# B&R Automation Studio project Panasonic_LinkaKapacitorov_A2021040 (part 2)

- Safety project (password-protected, skipped)

### Config.mprecipexml - AB1_CPU/mappServices/Config.mprecipexml
```
Element gRemPremenne (Type=mprecipexml)
```

### Config_1.mprecipexml - AB1_CPU/mappServices/Config_1.mprecipexml
```
Element gUzivatelXmlLink (Type=mprecipexml)
```

### Config_2.mprecipexml - AB1_CPU/mappServices/Config_2.mprecipexml
```
Element gRecipeXmlLink (Type=mprecipexml)
```

## Logical view

Binary libraries used (declarations not repeated): RUNTIME, OPERATOR, AsIecCon, astime, standard, AsBrStr, FileIO, sys_lib, AsSafety, DataObj, AsXml, CoTrace 5.14.0, AsZip, LoopConR 4.10.2, brsystem, dvframe, asstring, AsMath, AsTCP, MpRecipe 5.15.0, MpBase 5.15.0

### Global.typ - Global data types
```iecst
(********************************************************************
 * COPYRIGHT -- Microsoft
 ********************************************************************
 * File: Global.typ
 * Author: Martin
 * Created: February 11, 2016
 ********************************************************************
 * Global data types of project Zamazat_1
 ********************************************************************)
(**************Ovládanie tlačiarne**********************)

TYPE
	Client_typ : 	STRUCT  (*TCP Client Variables*)
		sStep : UINT; (*TCP Client Step Variable*)
		TcpOpen_0 : TcpOpen; (*AsTCP.TcpOpen FUB*)
		TcpClient_0 : TcpClient; (*AsTCP.TcpClient FUB*)
		TcpRecv_0 : TcpRecv; (*AsTCP.TcpRecv FUB*)
		TcpSend_0 : TcpSend; (*AsTCP.TcpSend FUB*)
		TcpIoctl_0 : TcpIoctl; (*AsTCP.TcpIoctl FUB*)
		TcpClose_0 : TcpClose; (*AsTCP.TcpClose FUB*)
		linger_opt : tcpLINGER_typ; (*AsTCP.tcpLINGER_typ*)
		recv_timeout : UDINT; (*receive timeout*)
		TcpOpen_timeout : UDINT;
		TcpClient_timeout : UDINT;
	END_STRUCT;
	Tlaciaren_typ : 	STRUCT
		Commands : TlaciarenCommands_typ;
		Status : TlaciarenStatus_typ;
		Data : TlaciarenData_typ;
	END_STRUCT;
	TlaciarenCommands_typ : 	STRUCT
		PosliSpravu : BOOL;
	END_STRUCT;
	TlaciarenStatus_typ : 	STRUCT
		PoruchaOtvoreniaKomunikacie : BOOL;
		PoruchaOdoslaniaDat : BOOL;
		PoruchaZatvoreniaKomunikacie : BOOL;
		PoruchaSpojenia_s_Tlaciarnou : BOOL;
		PoruchaPrijatiaDat : BOOL;
		PrislaSprava_s_Tlaciarne : BOOL;
	END_STRUCT;
	TlaciarenData_typ : 	STRUCT  (*Datatyp for global Variables*)
		Sprava_pre_Tlaciaren : STRING[4000]; (*Obsahuje posielane data pre tlačiareň v textovej podobe*)
		Odpoved_s_Tlaciarne : STRING[400]; (*Obsahuje odpoveď s tlačiarne*)
	END_STRUCT;
	EtiketaPanasonic_typ : 	STRUCT
		IdentificationNumber : STRING[10];
		ModelType : STRING[8];
		SupplierNumber : STRING[9];
		Country : STRING[2];
		Date : STRING[8];
		Counter : STRING[5];
		DataMetrix : STRING[31];
	END_STRUCT;
END_TYPE

(**********************RFID Čitačky*********************************************)

TYPE
	RFID_typ : 	STRUCT
		IN : RFID_IN_typ;
		OUT : RFID_OUT_typ;
		CMD : RFID_CMD_typ;
		STAV : RFID_STAV_typ;
		PAR : RFID_PAR_typ;
	END_STRUCT;
	RFID_IN_typ : 	STRUCT
		BYTE_IN : ARRAY[0..31]OF USINT;
		Bit_CP : BOOL;
		Bit_AA : BOOL;
		Bit_AE : BOOL;
		Bit_AF : BOOL;
		Bit_MT : BOOL;
		Bit_TO : BOOL;
		Old_Bit_TO : BOOL;
		Bit_HF : BOOL;
		Bit_BB : BOOL;
	END_STRUCT;
	RFID_OUT_typ : 	STRUCT
		BYTE_OUT : ARRAY[0..31]OF USINT;
		Bit_AV : BOOL;
		Bit_GR : BOOL;
		Bit_KA : BOOL;
		Bit_TI : BOOL;
	END_STRUCT;
	RFID_CMD_typ : 	STRUCT
		CitajDATA : BOOL;
		ZapisDATA : BOOL;
		CitaciuHlavu_VYPNI : BOOL;
	END_STRUCT;
	RFID_STAV_typ : 	STRUCT
		CitanieDat_OK : BOOL;
		CitanieDat_ERROR : BOOL;
		ZapisDat_OK : BOOL;
		ZapisDat_ERROR : BOOL;
		PritomnostCipu : BOOL;
	END_STRUCT;
	RFID_PAR_typ : 	STRUCT
		PrecitaneCisloPaletky : STRING[10];
		PrecitanyTypPaletky : STRING[10];
		Zadane_Cislo_Typ_Paletky : STRING[10]; (*Oddelovací znak "bodkočiarka"*)
		Precitane_Cislo_Typ_Paletky : STRING[10];
		PrecitaneCisloPaletky_POLE : ARRAY[0..9]OF USINT;
		ZadaneCisloPaletky_POLE : ARRAY[0..9]OF USINT;
	END_STRUCT;
END_TYPE

(**************************Ručná čitačka QR kódu******************************)

TYPE
	RS232_typ : 	STRUCT
		Command : RS232_Command_typ;
		Status : RS232_Status_typ;
		Step : USINT;
		FRM_xopen_0 : FRM_xopen;
		xopenConfig : XOPENCONFIG;
		FRM_read_0 : FRM_read;
		FRM_write_0 : FRM_write;
		FRM_rbuf_0 : FRM_rbuf;
		FRM_gbuf_0 : FRM_gbuf;
		FRM_robuf_0 : FRM_robuf;
		FRM_close_0 : FRM_close;
		PrecitaneData : STRING[80];
	END_STRUCT;
	RS232_Command_typ : 	STRUCT
		PosielajData : BOOL;
		PrimajData : BOOL;
		ZatvorKomunikaciu : BOOL;
		PotvrdeniePoruchy : BOOL;
	END_STRUCT;
	RS232_Status_typ : 	STRUCT
		PoruchaOtvoreniaKomunikacie : BOOL;
		PoruchaPriradeniaSEND_Buffera : BOOL;
		PoruchaUvolneniaSEND_Buffera : BOOL;
		PoruchaZatvoreniaKomunikacie : BOOL;
		PoruchaCitaniaDat : BOOL;
		PoruchaUvolneniaRECEIVE_Buffera : BOOL;
		PrimanieDat_OK : BOOL;
		PosielanieDat_OK : BOOL;
	END_STRUCT;
END_TYPE

(**************************Remanentne premenné********************************)

TYPE
	RemPremenne_typ : 	STRUCT
		VstupVytah_PozNavazania : UDINT;
		VstupVytah_PozVyvazania : UDINT;
		VystupVytah_PozNavazania : UDINT;
		VystupVytah_PozVyvazania : UDINT;
		PocetDniDoVymenyFiltra : UDINT;
	END_STRUCT;
END_TYPE

(***************Uzivatelia****************************)

TYPE
	ParametreUzivatelovTyp : 	STRUCT
		Meno : STRING[50];
		Heslo : STRING[50];
		UrovenUzivatela : UINT;
	END_STRUCT;
END_TYPE

(************Receptury*************************)

TYPE
	ParametreRecepturTyp : 	STRUCT
		NazovModelu : STRING[18];
		TypPaletky : STRING[4];
		Robot_CisloProgramu : USINT;
		Kamera_CisloProgramuQRkod : USINT;
		Kamera_CisloProgramuDMkod : USINT;
		Robot_PozLepenia_OffsetX : REAL;
		Robot_PozLepenia_OffsetY : REAL;
		Robot_PozLepenia_OffsetZ : REAL;
		RychlostDopravnikaPriCisteni : REAL;
	END_STRUCT;
END_TYPE

(**************************Safety***************************************************)

TYPE
	Safety_typ : 	STRUCT
		IN : Safety_IN_typ;
		OUT : Safety_OUT_typ;
		PAR : Safety_PAR_typ;
		STAV : Safety_STAV_typ;
		RESET_ZonyBunky : BOOL;
		RESET_ZonyCS : BOOL;
		RESET_ZonyVstupnehoVytahu : BOOL;
		RESET_ZonyVystupnehoVytahu : BOOL;
		RESET_DeadMan : BOOL;
		SpatnaVazba_ZonaBunky : BOOL;
		SpatnaVazba_ZonaCS : BOOL;
	END_STRUCT;
	Safety_IN_typ : 	STRUCT
		Robot_CS_CH1 : BOOL;
		Robot_CS_CH2 : BOOL;
		VyblokovanieSafety_CH1 : BOOL;
		VyblokovanieSafety_CH2 : BOOL;
		OvladaciPanel_CS_CH1 : BOOL;
		OvladaciPanel_CS_CH2 : BOOL;
		DopravnikNG_Bariera_CH1 : BOOL;
		DopravnikNG_Bariera_CH2 : BOOL;
		Snimac_ServisneDvere_CH1 : BOOL;
		Snimac_ServisneDvere_CH2 : BOOL;
		ZamkyBunky_CH1 : BOOL;
		ZamkyBunky_CH2 : BOOL;
		MutingRobota_CH1 : BOOL;
		MutingRobota_CH2 : BOOL;
		DeadMan_CH1 : BOOL;
		DeadMan_CH2 : BOOL;
		VstupnyVytah_MutingSnimac_CH1 : BOOL;
		VstupnyVytah_MutingSnimac_CH2 : BOOL;
		VstupnyVytah_Bariera_CH1 : BOOL;
		VstupnyVytah_Bariera_CH2 : BOOL;
		VstupnyVytah_CS_CH1 : BOOL;
		VstupnyVytah_CS_CH2 : BOOL;
		VystupnyVytah_MutingSnimac_CH1 : BOOL;
		VystupnyVytah_MutingSnimac_CH2 : BOOL;
		VystupnyVytah_Bariera_CH1 : BOOL;
		VystupnyVytah_Bariera_CH2 : BOOL;
		VystupnyVytah_CS_CH1 : BOOL;
		VystupnyVytah_CS_CH2 : BOOL;
	END_STRUCT;
	Safety_OUT_typ : 	STRUCT
		Zona_CS : BOOL;
		Zona_Bunky : BOOL;
		Zona_VstupnyVytah : BOOL;
		Zona_VystupnyVytah : BOOL;
	END_STRUCT;
	Safety_PAR_typ : 	STRUCT
		PAR_0 : USINT;
	END_STRUCT;
	Safety_STAV_typ : 	STRUCT
		SafetyPLC_Nabehlo : BOOL;
		ZonaCS_AKTIVNA : BOOL;
		ZonaBunky_Odblokovana : BOOL;
		ZamkyBunky_AKTIVNE : BOOL;
		ZonaBunky_AKTIVNA : BOOL;
		ZonaVstupnyVytah_Odblokovana : BOOL;
		ZonaVstupnyVytah_AKTIVNA : BOOL;
		ZonaVystupnyVytah_Odblokovana : BOOL;
		ZonaVystupnyVytah_AKTIVNA : BOOL;
		BarieraDopravnikaNG_AKTIVNA : BOOL;
		MutingRobota_AKTIVNY : BOOL;
		MutingBarieryVstupVytah_AKTIVNY : BOOL;
		MutingBarieryVystupVytah_AKTIVNY : BOOL;
		BarieraVstupVytahu_AKTIVNA : BOOL;
		BarieraVystupVytahu_AKTIVNA : BOOL;
		ServisneDvereTlaciarne_AKTIVNE : BOOL;
		CS_Robot_Odblokovany : BOOL;
		CS_OvlPanel_Odblokovany : BOOL;
		CS_VstupnyVytah_Odblokovany : BOOL;
		CS_VystupnyVytah_Odblokovany : BOOL;
		VyblokovanieSafety_AKTIVNE : BOOL;
		DeadMan_Odblokovany : BOOL;
		DeadMan_AKTIVNY : BOOL;
	END_STRUCT;
END_TYPE

(**************************Vizualizacia**********************************************)

TYPE
	Vizu_typ : 	STRUCT
		Language_Index : USINT;
		CisloAktualnejObrazovky : USINT;
		CisloZadanejObrazovky : USINT;
		TL_RezimAutomat : BOOL;
		TL_NavratPaletkyNG : BOOL;
		TL_ZamkniPredneDvere : BOOL;
		TL_ZamkniZadneDvere : BOOL;
		StavPracoviskaVstupVytah_Index : USINT;
		StavPracoviskaStopPredCist_Index : USINT;
		StavPracoviskaStopPoCist_Index : USINT;
		StavPracoviskaDoprCistenia_Index : USINT;
		StavPracoviskaStopEtiketov_Index : USINT;
		StavPracoviskaRobota_Index : USINT;
		StavPracoviskaDoprBunky_Index : USINT;
		StavPracoviskaStopDopNG_Index : USINT;
		StavPracoviskaStopVystDopr_Index : USINT;
		StavPracoviskaDoprVystup_Index : USINT;
		StavPracoviskaVystupVytah_Index : USINT;
		StavPracoviskaStopVratDopr_Index : USINT;
		StavPracoviskaDoprVrat_Index : USINT;
		StavZariadenia_Farba : USINT;
		StavZariadenia_Index : USINT;
		StavNGpaletky_Index : USINT;
		StavZmenyModelu_Index : USINT;
		StavZmenyModelu_Farba : USINT;
		TL_ZamokPredneDvere_DISABLE : BOOL;
		TL_ZamokZadneDvere_DISABLE : BOOL;
		TL_RezimManual_DISABLE : BOOL; (*0 - odomknuté, 1 - zamknuté*)
		TL_StartAutomat_DISABLE : BOOL;
		TL_UkoncenieCyklu_DISABLE : BOOL;
		TL_Reset_DISABLE : BOOL;
		TL_ZmenModel_DISABLE : BOOL;
		TL_PotvrdeniePaletky_NG_DISABLE : BOOL;
		TL_ZruseniePaletky_NG_DISABLE : BOOL;
		TL_OdparkujRobota_DISABLE : BOOL;
		ZmenaParametrov_DISABLE : BOOL;
		TL_BunkyRR_DISABLE : BOOL;
		TL_Ovl_Ionizatora_DISABLE : BOOL;
		TL_Ovl_DveriVstupVytahu_DISABLE : BOOL;
		Slider : USINT;
		FarbaTlacitkaAlarm_Index : BOOL;
		FarbaTlacitka_PotvrdPaletkuNG : BOOL;
		FarbaTlacitka_ZamokPredneDvere : USINT;
		FarbaTlacitka_ZamokZadneDvere : USINT;
		ZobrazSymbolAlarmu : BOOL;
		ZobrazHlasenie_ResetZariadenia : USINT;
		ZobrazHlasenie_PotvrdPaletkyNG : USINT;
		ZobrazHlasenie_NespravTypPaletky : USINT;
		ZobrazHlasenie_ZaaretujTlaciaren : USINT;
		ZobrazHlas_ZatvorSerDvereTlac : USINT;
		ZobrazHlasenie_TlaciarenOffline : USINT;
		ZobrazHlasenie_DochadzaPaska : USINT;
		PodsvietenieTlacitka_ResetCS : USINT;
		Nacitany_MODEL : STRING[18];
		Nacitany_LOT : STRING[11];
		NacitanieMODELU_DISABLE : BOOL;
		NacitanieLOTU_DISABLE : BOOL;
		NacitanieMODELU_IndexFarby : USINT;
		NacitanieLOTU_IndexFarby : USINT;
		OverNacitany_MODEL : BOOL;
		OverNacitany_LOT : BOOL;
		TL_VstupVytah_Homing_DISABLE : BOOL;
		TL_VstupVytah_Zdvih_DISABLE : BOOL;
		TL_VstupVytah_Doprav_DISABLE : BOOL;
		TL_VystupVytah_Homing_DISABLE : BOOL;
		TL_VystupVytah_Zdvih_DISABLE : BOOL;
		TL_VystupVytah_Doprav_DISABLE : BOOL;
		TL_Robot_CitanieQRkodu_DISABLE : BOOL;
		TL_Robot_CitanieDMkodu_DISABLE : BOOL;
		TL_Robot_OdoberEtiketu_DISABLE : BOOL;
		ZadavanieKorekciiRobota_DISABLE : BOOL;
		VolbyRezimov_DISABLE : BOOL;
		IndexSuradnicovehoSystemuPaletky : USINT;
		IndexFarbyStavuFiltrov : USINT;
		IndexStavuFiltrov : USINT;
		IndexStavuPasky : USINT;
		IndexStavuLadenieKamery : USINT;
		IndexStavuLadenieKamery_Farba : USINT;
		ZobrazSymbolCS_VstupVytah : USINT;
		ZobrazSymbolCS_VystupVytah : USINT;
		ZobrazSymbolCS_Panel : USINT;
		ZobrazSymbolCS_Robot : USINT;
	END_STRUCT;
END_TYPE

(**************************Linka************************************************)

TYPE
	Linka_typ : 	STRUCT
		IN : Linka_IN_typ;
		OUT : Linka_OUT_typ;
		PAR : Linka_PAR_typ;
		STAV : Linka_STAV_typ;
		Automat : BOOL;
		Manual : BOOL;
		Reset : BOOL;
		KoniecCyklu : BOOL;
		Majak_HukackaON : BOOL;
		CitackaQRkodu_AKTIVNA : BOOL;
		ZmenModel : BOOL;
		VymenaFiltrovPotvrdena : BOOL;
		Rezim_BezTlaceEtikety : BOOL;
		Rezim_BezKomunikacie : BOOL;
		Rezim_BezCistenia : BOOL;
		Rezim_Priechodny : BOOL;
		Rezim_Testovania : BOOL;
		ResetNapajaniaKamery : BOOL;
	END_STRUCT;
	Linka_IN_typ : 	STRUCT
		PrepatovaOchrana_OK : BOOL; (*1 - OK*)
		PoruchaNapajaniaMenicov : BOOL; (*1 - OK*)
		SpatnaVazba_ZonaCS : BOOL; (*1 - OK*)
		SpatnaVazba_ZonaVstupVytah : BOOL; (*1 - OK*)
		SpatnaVazba_ZonaVystupVytah : BOOL; (*1 - OK*)
		SpatnaVazba_ZonaBunky : BOOL; (*1 - OK*)
		SpatnaVazba_VentilTerminal_SQ1 : BOOL;
		SpatnaVazba_VentilTerminal_SQ2 : BOOL;
		PredneDvereZavrete_EZ1 : BOOL;
		ZadneDvereZavrete_EZ2 : BOOL;
		SmartKamera_IN0_CAM1 : BOOL;
		SmartKamera_IN1_CAM1 : BOOL;
		TlakVzduchu_OK_S2 : BOOL;
		IonJednotka_MachineON_RJ1 : BOOL;
		IonJednotka_Error_Sumary_RJ1 : BOOL;
		IonJednotka_Error_Filter1_RJ1 : BOOL;
		IonJednotka_Error_Filter2_RJ1 : BOOL;
		IonJednotka_Error_Motor_RJ1 : BOOL;
		IonJednotka_Error_Network_RJ1 : BOOL;
		IonJednotka_Error_HighVolt_RJ1 : BOOL;
		IonJednotka_Error_ComAirTC1_RJ1 : BOOL;
		IonJednotka_Error_ComAirTC2_RJ1 : BOOL;
		IonJednotka_Error_VolumeFlow_RJ1 : BOOL;
		IonJednotka_Error_TCcontrol_RJ1 : BOOL;
		IonJednotka_Error_Inverter_RJ1 : BOOL;
		IonJednotka_PoruchaNapajania : BOOL;
		SnimacRotacieHornTrysiek_1_IS7 : BOOL;
		SnimacRotacieHornTrysiek_2_IS8 : BOOL;
		SnimacRotacieHornTrysiek_3_IS9 : BOOL;
		SnimacRotacieHornTrysiek_4_IS10 : BOOL;
		SnimacRotacieSpodTrysiek_1_IS11 : BOOL;
		SnimacRotacieSpodTrysiek_2_IS12 : BOOL;
		SnimacRotacieSpodTrysiek_3_IS13 : BOOL;
	END_STRUCT;
	Linka_OUT_typ : 	STRUCT
		Majak_ZeleneSvetlo : BOOL;
		Majak_ZlteSvetlo : BOOL;
		Majak_CerveneSvetlo : BOOL;
		Majak_Hukacka : BOOL;
		PredneDvere_Zamkni_EZ1 : BOOL;
		ZadneDvere_Zamkni_EZ2 : BOOL;
		OsvetlenieBunky_Zapni : BOOL;
		SmartKamera_OUT0_CAM1 : BOOL;
		SmartKamera_OUT1_CAM1 : BOOL;
		VT1_PowerlinkOUTPUTS : ARRAY[0..3]OF USINT;
		IonJednotka_START : BOOL;
		IonJednotka_RESET : BOOL;
		IonJednotka_AIR : BOOL;
		Vzduchotechnika_START : BOOL;
		Rele_ResetNapajaniaKamery : BOOL;
	END_STRUCT;
	Linka_PAR_typ : 	STRUCT
		Zvoleny_MODEL : STRING[18];
		Zvoleny_LOT : STRING[11];
		Zvoleny_TypPaletky : STRING[10];
		IndexZvoleneReceptury : USINT;
		Zvolene_CisloProgramuRobota : USINT;
		Zvolene_KamCisloProg_QRkod : USINT;
		Zvolene_KamCisloProg_DMkod : USINT;
		Zvolena_PozLepenia_OffsetX : REAL;
		Zvolena_PozLepenia_OffsetY : REAL;
		Zvolena_PozLepenia_OffsetZ : REAL;
		Zvolena_RychlostDopravPriCisteni : REAL;
	END_STRUCT;
	Linka_STAV_typ : 	STRUCT
		Automat : BOOL;
		Manual : BOOL;
		PoINIT : BOOL;
		READY_TO_START : BOOL;
		UkoncenieCyklu_BUSY : BOOL;
		Hardware_OK : BOOL;
		PrebiehaZmenaModelu : BOOL;
		PoruchaOtacaniaTrysiek : BOOL;
		FiltreIonizacnejJednotkyZanesene : BOOL;
		IonizacnaJednotka_BUSY : BOOL;
		Dopravniky_PAUZA : BOOL;
	END_STRUCT;
END_TYPE

(**************Stav hardware*****************************)

TYPE
	Hardware_STAV_typ : 	STRUCT
		KartaAB2_ProfinetMaster_OK : BOOL;
		KartaAB3_SafetyMaster_OK : BOOL;
		KartaAB4_SafetyDI_OK : BOOL;
		KartaAB5_16DI_OK : BOOL;
		KartaAB6_16DI_OK : BOOL;
		KartaAB7_16DI_OK : BOOL;
		KartaAB8_16DO_OK : BOOL;
		KartaAB9_16DO_OK : BOOL;
		KartaAB10_X2X_OK : BOOL;
		ModulDI1_16DI_OK : BOOL;
		ModulDI2_16DI_OK : BOOL;
		ModulDI3_8DI_OK : BOOL;
		ModulSI1_4SI_OK : BOOL;
		ModulSI2_4SI_OK : BOOL;
		Komunikacia_Robot_OK : BOOL;
		Komunikacia_Kamera_OK : BOOL;
		Komunikacia_RFIDModul_OK : BOOL;
		Komunikacia_VentTerminal_OK : BOOL;
		Komunikacia_MeniceFM_OK : BOOL;
		Komunikacia_Panasonic_OK : BOOL;
	END_STRUCT;
END_TYPE

(***************VstupnyVytah*************************************)

TYPE
	VstupnyVytah_typ : 	STRUCT
		IN : VstupnyVytah_IN_typ;
		OUT : VstupnyVytah_OUT_typ;
		PAR : VstupnyVytah_PAR_typ;
		STAV : VstupnyVytah_STAV_typ;
		Automat : BOOL;
		Manual : BOOL;
		Reset : BOOL;
		KoniecCyklu : BOOL;
		MenicZdvihu_FM2 : RiadenieFM;
		RR_Dopravnik_VPRED : BOOL;
		RR_Dopravnik_VZAD : BOOL;
	END_STRUCT;
	VstupnyVytah_IN_typ : 	STRUCT
		RiadenieDopravnika_OK_ELR1 : BOOL;
		TeplotaMotora_OK_M1 : BOOL; (*1 - OK*)
		StavMenicaZdvihu_OK_FM2 : BOOL; (*1 - OK*)
		BannerPotvrdeny_IOS1 : BOOL;
		DvereVytahuOtvorene_MS1 : BOOL;
		DvereVytahuZatvorene_MS2 : BOOL;
		PrechodDopravnikaVytahu_OS1 : BOOL;
		PritomnostPaletky_IS3 : BOOL;
		PritomnostProduktu_OS2 : BOOL;
		ReferencnySnimacZdvihu : BOOL; (*Preposielané z FM cez komunikáciu*)
		SpodnyLimitZdvihu : BOOL; (*Preposielané z FM cez komunikáciu*)
		HornyLimitZdvihu : BOOL; (*Preposielané z FM cez komunikáciu*)
	END_STRUCT;
	VstupnyVytah_OUT_typ : 	STRUCT
		Dopravnik_ChodVPRED_ELR1 : BOOL;
		Dopravnik_ChodVZAD_ELR1 : BOOL;
		Banner_ZelenaLED_IOS1 : BOOL;
		Banner_CervenaLED_IOS1 : BOOL;
		DvereVytahu_OTVOR_YV002 : BOOL;
		DvereVytahu_ZATVOR_YV001 : BOOL;
	END_STRUCT;
	VstupnyVytah_PAR_typ : 	STRUCT
		Zdvih_ZadanaPozicia : UDINT;
		Zdvih_ZadanaRychlost : REAL;
		Zdvih_ZadanaJoggRychlost : REAL;
	END_STRUCT;
	VstupnyVytah_STAV_typ : 	STRUCT
		PoINIT : BOOL;
		Zdvih_AktualnaPozicia : UDINT;
		Zdvih_AktualnaRychlost : REAL;
		Zdvih_HomingOK : BOOL;
		Zdvih_BUSY : BOOL;
		Homing_BUSY : BOOL;
		Zdvih_PoziciaDosiahnuta : BOOL;
		PrebiehaVyvazaniePaletky : BOOL;
		VytahNapolohovany : BOOL;
		ObsluhaPotvrdilaBanner : BOOL;
	END_STRUCT;
END_TYPE

(***************StoperPredCistenim*************************************)

TYPE
	StoperPredCistenim_typ : 	STRUCT
		IN : StoperPredCistenim_IN_typ;
		OUT : StoperPredCistenim_OUT_typ;
		PAR : StoperPredCistenim_PAR_typ;
		STAV : StoperPredCistenim_STAV_typ;
		Automat : BOOL;
		Manual : BOOL;
		Reset : BOOL;
		KoniecCyklu : BOOL;
	END_STRUCT;
	StoperPredCistenim_IN_typ : 	STRUCT
		PritomnostPaletky_IS4 : BOOL;
	END_STRUCT;
	StoperPredCistenim_OUT_typ : 	STRUCT
		StoperZASUN_YV005 : BOOL;
	END_STRUCT;
	StoperPredCistenim_PAR_typ : 	STRUCT
		PAR_0 : USINT;
	END_STRUCT;
	StoperPredCistenim_STAV_typ : 	STRUCT
		PoINIT : BOOL;
		PrebiehaVyvazaniePaletky : BOOL;
	END_STRUCT;
END_TYPE

(***************StoperPoCisteni*************************************)

TYPE
	StoperPoCisteni_typ : 	STRUCT
		IN : StoperPoCisteni_IN_typ;
		OUT : StoperPoCisteni_OUT_typ;
		PAR : StoperPoCisteni_PAR_typ;
		STAV : StoperPoCisteni_STAV_typ;
		Automat : BOOL;
		Manual : BOOL;
		Reset : BOOL;
		KoniecCyklu : BOOL;
	END_STRUCT;
	StoperPoCisteni_IN_typ : 	STRUCT
		PritomnostPaletky_IS6 : BOOL;
		ZaplnenieBuffera_IS5 : BOOL;
	END_STRUCT;
	StoperPoCisteni_OUT_typ : 	STRUCT
		StoperZASUN_YV006 : BOOL;
	END_STRUCT;
	StoperPoCisteni_PAR_typ : 	STRUCT
		PAR_0 : USINT;
	END_STRUCT;
	StoperPoCisteni_STAV_typ : 	STRUCT
		PoINIT : BOOL;
		PrebiehaVyvazaniePaletky : BOOL;
	END_STRUCT;
END_TYPE

(***************DopravnikCistenia*************************************)

TYPE
	DopravCistenia_typ : 	STRUCT
		IN : DopravCistenia_IN_typ;
		OUT : DopravCistenia_OUT_typ;
		PAR : DopravCistenia_PAR_typ;
		STAV : DopravCistenia_STAV_typ;
		Automat : BOOL;
		Manual : BOOL;
		Reset : BOOL;
		KoniecCyklu : BOOL;
		MenicDopravnika_FM1 : RiadenieFM;
		RR_Chod_VPRED : BOOL;
		RR_Chod_VZAD : BOOL;
		Dopravnik_RUN : BOOL;
	END_STRUCT;
	DopravCistenia_IN_typ : 	STRUCT
		StavMenica_OK_FM1 : BOOL; (*1 - OK*)
	END_STRUCT;
	DopravCistenia_OUT_typ : 	STRUCT
		New_Member : USINT;
	END_STRUCT;
	DopravCistenia_PAR_typ : 	STRUCT
		ZadanaRychlost : REAL;
		ZadanaJoggRychlost : REAL;
	END_STRUCT;
	DopravCistenia_STAV_typ : 	STRUCT
		PoINIT : BOOL;
		AktualnaRychlost : REAL;
		BUSY : BOOL;
	END_STRUCT;
END_TYPE

(***************DopravnikBunky*************************************)

TYPE
	DopravBunky_typ : 	STRUCT
		IN : DopravBunky_IN_typ;
		OUT : DopravBunky_OUT_typ;
		PAR : DopravBunky_PAR_typ;
		STAV : DopravBunky_STAV_typ;
		Automat : BOOL;
		Manual : BOOL;
		Reset : BOOL;
		KoniecCyklu : BOOL;
	END_STRUCT;
	DopravBunky_IN_typ : 	STRUCT
		RiadenieDopravnika_OK_ELR4 : BOOL;
		TeplotaMotora_OK_M4 : BOOL; (*1 - OK*)
	END_STRUCT;
	DopravBunky_OUT_typ : 	STRUCT
		Dopravnik_ChodVPRED_ELR4 : BOOL;
	END_STRUCT;
	DopravBunky_PAR_typ : 	STRUCT
		PAR_0 : USINT;
	END_STRUCT;
	DopravBunky_STAV_typ : 	STRUCT
		PoINIT : BOOL;
	END_STRUCT;
END_TYPE

(***************StoperEtiketovania*************************************)

TYPE
	StoperEtiketovania_typ : 	STRUCT
		IN : StoperEtiketovania_IN_typ;
		OUT : StoperEtiketovania_OUT_typ;
		PAR : StoperEtiketovania_PAR_typ;
		STAV : StoperEtiketovania_STAV_typ;
		Automat : BOOL;
		Manual : BOOL;
		Reset : BOOL;
		KoniecCyklu : BOOL;
		RR_VytlacEtiketu : BOOL;
		OdosliDataDoPanasonicu : BOOL;
		RR_ZacentrujPaletku : BOOL;
		RR_OdcentrujPaletku : BOOL;
	END_STRUCT;
	StoperEtiketovania_IN_typ : 	STRUCT
		Tlaciaren_KoniecEtikiet : BOOL;
		Tlaciaren_KoniecPasky : BOOL;
		Tlaciaren_Porucha : BOOL;
		Tlaciaren_KoniecTlace : BOOL;
		Tlaciaren_Offline : BOOL;
		Tlaciaren_Dispending : BOOL;
		PritomnostPaletky_IS16 : BOOL;
		Centrovanie_HornaPoloha_IS18 : BOOL;
		Centrovanie_SpodnaPoloha_IS17 : BOOL;
		SuflikTlaciarne_LS_IS23 : BOOL;
		SuflikTlaciarne_PS_IS22 : BOOL;
	END_STRUCT;
	StoperEtiketovania_OUT_typ : 	STRUCT
		Tlaciaren_VytlacEtiketu : BOOL;
		Tlaciaren_VytlacZnovaEtiketu : BOOL;
		Centrovanie_VYSUN_YV003 : BOOL;
		Centrovanie_ZASUN_YV004 : BOOL;
		StoperZASUN_YV007 : BOOL;
	END_STRUCT;
	StoperEtiketovania_PAR_typ : 	STRUCT
		TypPaletky_RucneVytlacEtikety : STRING[3];
	END_STRUCT;
	StoperEtiketovania_STAV_typ : 	STRUCT
		PoINIT : BOOL;
		PrebiehaVyvazaniePaletky : BOOL;
		TlaciarenZaaretovana : BOOL;
		Etiketovanie_BUSY : BOOL;
		VyvazamPaletkuNG : BOOL;
		AlarmTextPaletkyNG : STRING[30];
		Warning : BOOL;
	END_STRUCT;
END_TYPE

(***************Robot************************************)

TYPE
	Robot_typ : 	STRUCT
		IN : Robot_IN_typ;
		OUT : Robot_OUT_typ;
		KOM_IN : RobotKOM_IN_typ;
		KOM_OUT : RobotKOM_OUT_typ;
		PAR : Robot_PAR_typ;
		STAV : Robot_STAV_typ;
		Automat : BOOL;
		Manual : BOOL;
		Reset : BOOL;
		KoniecCyklu : BOOL;
		PrisavanieEtikety_ZAPNI : BOOL;
		Odparkovanie : BOOL;
		RR_PresunPoziciaCitaniaQRkodu : BOOL;
		RR_PresunPoziciaCitaniaDMkodu : BOOL;
		RR_PresunPoziciaOdobratiaEtikety : BOOL;
		RR_PresunPoziciaNalepeniaEtikety : BOOL;
	END_STRUCT;
	Robot_IN_typ : 	STRUCT
		PrisatieEtikety_OK_S1 : BOOL;
	END_STRUCT;
	Robot_OUT_typ : 	STRUCT
		PrisavanieEtikety_ZAPNI_YV013 : BOOL;
		PrisavanieEtikety_VYPNI_YV014 : BOOL;
	END_STRUCT;
	Robot_PAR_typ : 	STRUCT
		New_Member : USINT;
	END_STRUCT;
	Robot_STAV_typ : 	STRUCT
		PoINIT : BOOL;
	END_STRUCT;
	RobotKOM_IN_typ : 	STRUCT
		Stav_RobotOdparkovany : BOOL;
		Stav_RobotDrziEtiketu : BOOL;
		Stav_RobotCinnostUkoncena : BOOL;
		Stav_MotoryON : BOOL;
		Stav_MotoryOFF : BOOL;
		Stav_ProgramRUN : BOOL;
		Stav_RezimAUTOMAT : BOOL;
		Stav_RobotCS : BOOL;
		Stav_VystupyZresetovane : BOOL;
		Stav_ZonaNavratuRobota_OK : BOOL;
		Stav_ZonaNavratuRobota_NG : BOOL;
		Stav_PoruchaRobota : BOOL;
		Profinet_PLC_INPUTS : ARRAY[0..63]OF USINT;
	END_STRUCT;
	RobotKOM_OUT_typ : 	STRUCT
		ZapniMotory : BOOL;
		VypniMotory : BOOL;
		PP_na_Main : BOOL;
		Reset_CS : BOOL;
		StartProgramu : BOOL;
		StartProgramuMain : BOOL;
		StopProgramu : BOOL;
		OdparkujRobota : BOOL;
		ServisnaPozicia : BOOL;
		ZahodEtiketu : BOOL;
		NalepEtiketu : BOOL;
		PresunDoVychodiskovejPozicie : BOOL;
		PresunDoMutingPozicie : BOOL;
		PresunDoPozicieOdobratiaEtikety : BOOL;
		PresunDoPoziceKontrolyEtikety : BOOL;
		PresunDoPoziceKontrEtiketyPriamo : BOOL;
		PresunDoPozicieKontrolyIntStitku : BOOL;
		CitanieStitkuUkoncene : BOOL;
		UkoncenieCykluRobota : BOOL;
		CisloProduktu : USINT;
		LepenieStitku_OffsetX : USINT;
		LepenieStitku_OffsetY : USINT;
		LepenieStitku_OffsetZ : USINT;
		LepenieStitku_ZnamienkoOffsetX : BOOL;
		LepenieStitku_ZnamienkoOffsetY : BOOL;
		LepenieStitku_ZnamienkoOffsetZ : BOOL;
		Profinet_PLC_OUTPUTS : ARRAY[0..63]OF USINT;
	END_STRUCT;
END_TYPE

(***************StoperDopravnikaNG*************************************)

TYPE
	StoperDopravnikaNG_typ : 	STRUCT
		IN : StoperDopravnikaNG_IN_typ;
		OUT : StoperDopravnikaNG_OUT_typ;
		PAR : StoperDopravnikaNG_PAR_typ;
		STAV : StoperDopravnikaNG_STAV_typ;
		Automat : BOOL;
		Manual : BOOL;
		Reset : BOOL;
		KoniecCyklu : BOOL;
		RR_Dopravnik_VPRED : BOOL;
		RR_Dopravnik_VZAD : BOOL;
	END_STRUCT;
	StoperDopravnikaNG_IN_typ : 	STRUCT
		Stoper_PritomnostPaletky_IS15 : BOOL;
		Dopravnik_PritomnostPaletky_OS4 : BOOL;
		Dopravnik_PritomnostProduktu_OS3 : BOOL;
		Centrovanie_HornaPoloha_IS19 : BOOL;
		Centrovanie_StrednaPoloha_IS20 : BOOL;
		Centrovanie_SpodnaPoloha_IS21 : BOOL;
		RiadenieDopravnika_OK_ELR3 : BOOL;
		TeplotaMotora_OK_M3 : BOOL; (*1 - OK*)
	END_STRUCT;
	StoperDopravnikaNG_OUT_typ : 	STRUCT
		NatlakujTlmicPaletky_YV008 : BOOL;
		Centrovanie_VYSUN_YV009 : BOOL; (*Transport na NG dopravník*)
		Centrovanie_ZASUN_YV010 : BOOL; (*Transport na výstupný dopravník*)
		Dopravnik_ChodVPRED_ELR3 : BOOL;
		Dopravnik_ChodVZAD_ELR3 : BOOL;
	END_STRUCT;
	StoperDopravnikaNG_PAR_typ : 	STRUCT
		New_Member : USINT;
	END_STRUCT;
	StoperDopravnikaNG_STAV_typ : 	STRUCT
		PoINIT : BOOL;
		ObsluhaPotvrdilaPaletkuNG : BOOL;
		ObsluhaPotvrdilaZrusPaletkyNG : BOOL;
		PrebiehaVyvazaniePaletky : BOOL;
		PaletkaNaKonciDopravnika_NG : BOOL;
		DopravnikNG_BUSY : BOOL;
	END_STRUCT;
END_TYPE

(***************VystupnyDopravnik*************************************)

TYPE
	VystupnyDopravnik_typ : 	STRUCT
		IN : VystupnyDopravnik_IN_typ;
		OUT : VystupnyDopravnik_OUT_typ;
		PAR : VystupnyDopravnik_PAR_typ;
		STAV : VystupnyDopravnik_STAV_typ;
		Automat : BOOL;
		Manual : BOOL;
		Reset : BOOL;
		KoniecCyklu : BOOL;
	END_STRUCT;
	VystupnyDopravnik_IN_typ : 	STRUCT
		RiadenieDopravnika_OK_ELR5 : BOOL;
		TeplotaMotora_OK_M5 : BOOL;
	END_STRUCT;
	VystupnyDopravnik_OUT_typ : 	STRUCT
		Dopravnik_ChodVPRED_ELR5 : BOOL;
	END_STRUCT;
	VystupnyDopravnik_PAR_typ : 	STRUCT
		PAR_0 : USINT;
	END_STRUCT;
	VystupnyDopravnik_STAV_typ : 	STRUCT
		PoINIT : BOOL;
	END_STRUCT;
END_TYPE

(***************StoperVystupDopravnika*************************************)

TYPE
	StoperVystupDopravnika_typ : 	STRUCT
		IN : StoperVystupDopravnika_IN_typ;
		OUT : StoperVystupDopravnika_OUT_typ;
		PAR : StoperVystupDopravnika_PAR_typ;
		STAV : StoperVystupDopravnika_STAV_typ;
		Automat : BOOL;
		Manual : BOOL;
		Reset : BOOL;
		KoniecCyklu : BOOL;
	END_STRUCT;
	StoperVystupDopravnika_IN_typ : 	STRUCT
		PritomnostPaletky_IS27 : BOOL;
		ZaplnenieBuffera_IS28 : BOOL;
	END_STRUCT;
	StoperVystupDopravnika_OUT_typ : 	STRUCT
		StoperZASUN_YV011 : BOOL;
	END_STRUCT;
	StoperVystupDopravnika_PAR_typ : 	STRUCT
		PAR_0 : USINT;
	END_STRUCT;
	StoperVystupDopravnika_STAV_typ : 	STRUCT
		PoINIT : BOOL;
		PrebiehaVyvazaniePaletky : BOOL;
	END_STRUCT;
END_TYPE

(***************VystupnyVytah*************************************)

TYPE
	VystupnyVytah_typ : 	STRUCT
		IN : VystupnyVytah_IN_typ;
		OUT : VystupnyVytah_OUT_typ;
		PAR : VystupnyVytah_PAR_typ;
		STAV : VystupnyVytah_STAV_typ;
		Automat : BOOL;
		Manual : BOOL;
		Reset : BOOL;
		KoniecCyklu : BOOL;
		MenicZdvihu_FM3 : RiadenieFM;
		RR_Dopravnik_VPRED : BOOL;
		RR_Dopravnik_VZAD : BOOL;
	END_STRUCT;
	VystupnyVytah_IN_typ : 	STRUCT
		RiadenieDopravnika_OK_ELR6 : BOOL;
		TeplotaMotora_OK_M6 : BOOL; (*1 - OK*)
		StavMenicaZdvihu_OK_FM3 : BOOL; (*1 - OK*)
		BannerPotvrdeny_IOS2 : BOOL;
		PritomnostPaletky_IS26 : BOOL;
		PritomnostProduktu_OS5 : BOOL;
		PrechodDopravnikaVytahu_OS6 : BOOL;
		ReferencnySnimacZdvihu : BOOL; (*Preposielané z FM cez komunikáciu*)
		SpodnyLimitZdvihu : BOOL; (*Preposielané z FM cez komunikáciu*)
		HornyLimitZdvihu : BOOL; (*Preposielané z FM cez komunikáciu*)
		SpodnySpomalovaciSnimac : BOOL;
		HornySpomalovaciSnimac : BOOL;
	END_STRUCT;
	VystupnyVytah_OUT_typ : 	STRUCT
		Dopravnik_ChodVPRED_ELR6 : BOOL;
		Dopravnik_ChodVZAD_ELR6 : BOOL;
		Banner_ZelenaLED_IOS2 : BOOL;
		Banner_CervenaLED_IOS2 : BOOL;
	END_STRUCT;
	VystupnyVytah_PAR_typ : 	STRUCT
		Zdvih_ZadanaPozicia : UDINT;
		Zdvih_ZadanaRychlost : REAL;
		Zdvih_ZadanaJoggRychlost : REAL;
	END_STRUCT;
	VystupnyVytah_STAV_typ : 	STRUCT
		PoINIT : BOOL;
		Zdvih_AktualnaPozicia : UDINT;
		Zdvih_AktualnaRychlost : REAL;
		Zdvih_HomingOK : BOOL;
		Zdvih_BUSY : BOOL;
		Homing_BUSY : BOOL;
		Zdvih_PoziciaDosiahnuta : BOOL;
		PrebiehaVyvazaniePaletky : BOOL;
		VytahNapolohovany : BOOL;
	END_STRUCT;
END_TYPE

(***************VratnyDopravnik*************************************)

TYPE
	VratnyDopravnik_typ : 	STRUCT
		IN : VratnyDopravnik_IN_typ;
		OUT : VratnyDopravnik_OUT_typ;
		PAR : VratnyDopravnik_PAR_typ;
		STAV : VratnyDopravnik_STAV_typ;
		Automat : BOOL;
		Manual : BOOL;
		Reset : BOOL;
		KoniecCyklu : BOOL;
	END_STRUCT;
	VratnyDopravnik_IN_typ : 	STRUCT
		RiadenieDopravnika_OK_ELR2 : BOOL;
		TeplotaMotora_OK_M2 : BOOL;
	END_STRUCT;
	VratnyDopravnik_OUT_typ : 	STRUCT
		Dopravnik_ChodVPRED_ELR2 : BOOL;
	END_STRUCT;
	VratnyDopravnik_PAR_typ : 	STRUCT
		PAR_0 : USINT;
	END_STRUCT;
	VratnyDopravnik_STAV_typ : 	STRUCT
		PoINIT : BOOL;
	END_STRUCT;
END_TYPE

(***************StoperVratnehoDopravnika*************************************)

TYPE
	StoperVratDopravnika_typ : 	STRUCT
		IN : StoperVratDopravnika_IN_typ;
		OUT : StoperVratDopravnika_OUT_typ;
		PAR : StoperVratDopravnika_PAR_typ;
		STAV : StoperVratDopravnika_STAV_typ;
		Automat : BOOL;
		Manual : BOOL;
		Reset : BOOL;
		KoniecCyklu : BOOL;
	END_STRUCT;
	StoperVratDopravnika_IN_typ : 	STRUCT
		PritomnostPaletky_IS14 : BOOL;
	END_STRUCT;
	StoperVratDopravnika_OUT_typ : 	STRUCT
		StoperZASUN_YV012 : BOOL;
	END_STRUCT;
	StoperVratDopravnika_PAR_typ : 	STRUCT
		PAR_0 : USINT;
	END_STRUCT;
	StoperVratDopravnika_STAV_typ : 	STRUCT
		PoINIT : BOOL;
		PrebiehaVyvazaniePaletky : BOOL;
	END_STRUCT;
END_TYPE

(*****************Kamera*****************************************)

TYPE
	CAM_typ : 	STRUCT
		CMD : CAM_CMD_typ;
		PAR : CAM_PAR_typ;
		STAV : CAM_STAV_typ;
		RESULT : CAM_RESULTS_typ;
		Profinet_InterEtiketaQRznaky : ARRAY[0..63]OF USINT;
		Profinet_ZakazEtiketaDMznaky : ARRAY[0..63]OF USINT;
		Profinet_PLC_INPUTS : ARRAY[0..10]OF USINT;
		Profinet_PLC_OUTPUTS : USINT;
	END_STRUCT;
	CAM_CMD_typ : 	STRUCT
		Triger : BOOL;
	END_STRUCT;
	CAM_PAR_typ : 	STRUCT
		ZadaneCisloProgramu : USINT;
	END_STRUCT;
	CAM_STAV_typ : 	STRUCT
		BUSY : BOOL;
		SWITCH : BOOL;
		READY : BOOL;
		Results_READY : BOOL;
		AktualneCisloProgramu : USINT;
		RUN_Counter : USINT;
		Old_Hodnota_RUN_Counter : USINT;
	END_STRUCT;
	CAM_RESULTS_typ : 	STRUCT
		ZakazEtiketa_DMkod_OK : BOOL;
		InternaEtiketa_QRkod_OK : BOOL;
		ZakazEtiketa_PritomnZnakov_OK : BOOL;
		BielyPatern_OK : BOOL;
		InternaEtiketa_ZnakyQRkodu : STRING[64];
		ZakazEtiketa_ZnakyDMkodu : STRING[64];
	END_STRUCT;
END_TYPE

(*************Parametre paletky*********************)

TYPE
	Paletka_typ : 	STRUCT
		StavPaletky : STRING[2]; (*OK, NG, PR*)
		CisloPaletky : STRING[4]; (*Prečítané čitačkou RFID*)
		TypPaletky : STRING[4]; (*Prečítané čitačkou RFID*)
		NazovPaletky : STRING[10]; (*Vyskladaný z čísla paletky a typu paletky*)
		NazovModelu : STRING[18]; (*Načítaný z čitačky*)
		CisloLOT : STRING[20]; (*Načítaný z čitačky*)
		Robot_CisloProgramu : USINT;
		Kamera_CisloProgramu_QRkod : USINT;
		Kamera_CisloProgramu_DMkod : USINT;
		TypVyroby : STRING[1]; (*Vždy druhý znak z Lotu  0 - Regular, S - Sample, P - Preproduct, E - Early evaluation *)
		InternySerialNumber : STRING[48]; (*Prečítaný z kapacitora*)
		ZakaznickeCislo : STRING[49]; (*Prijaté zo servera*)
		PrecitaneZnakyZakaznickehoDMkodu : STRING[49]; (*Prečítané zo zákaznickej etikety*)
		ReturnProcessName : STRING[30];
		Cistenie_DONE : BOOL;
		StavCistenia : STRING[2]; (*OK alebo NG*)
		NalepenieEtikety_DONE : BOOL;
		StavNalepeniaEtikety : STRING[2]; (*OK alebo NG*)
		StavCitania_InternehoQRkodu : STRING[2]; (*OK alebo NG*)
		StavCitania_ZakaznickehoDMkodu : STRING[2]; (*OK alebo NG*)
		StavCitania_KontrolaZnakov : STRING[2]; (*OK alebo NG*)
		StavPorovnaniaDMkoduZoServerom : STRING[2]; (*OK alebo NG*)
		StavKontrolyBielehoPaternu : STRING[2]; (*OK alebo NG*)
		StavKomunikacie_DONE : BOOL;
	END_STRUCT;
END_TYPE

(*************Historia výroby************************)

TYPE
	HystoriaVyroby_typ : 	STRUCT
		NazovModelu : STRING[18];
		NazovLOTU : STRING[11];
		PocetVyrobenychKusov_OK : REAL;
		PocetVyrobenychKusov_NG : REAL;
		Pomer_OK_kusov_IDR : REAL;
	END_STRUCT;
END_TYPE

(*************Motohodiny****************************)

TYPE
	Motohodiny_typ : 	STRUCT
		Milisekundy : UINT;
		Sekundy : USINT;
		Minuty : USINT;
		Hodiny : USINT;
		Dny : UDINT;
		CelkovyPocetHodin : UDINT;
		START : BOOL;
		RESET : BOOL;
	END_STRUCT;
END_TYPE
```

### Global.var - Global variables
```iecst
(********************************************************************
 * COPYRIGHT -- Microsoft
 ********************************************************************
 * File: Global.var
 * Author: Martin
 * Created: February 11, 2016
 ********************************************************************
 * Global variables of project Zamazat_1
 ********************************************************************)
VAR
	Pocitadlo : UDINT := 0;
	Prisavka_ON : BOOL := FALSE;
END_VAR
(******************RFID čitačky**********************)
VAR
	RFID_Hlava_1 : RFID_typ;
	SC_Hlava_1 : SequenceControlTyp;
	RFID_Hlava_2 : RFID_typ;
	SC_Hlava_2 : SequenceControlTyp;
	RFID_Hlava_3 : RFID_typ;
	SC_Hlava_3 : SequenceControlTyp;
	RFID_Hlava_4 : RFID_typ;
	SC_Hlava_4 : SequenceControlTyp;
END_VAR
(**************Ručná čítačka QR kódu************)
VAR
	RucCitackaQR : RS232_typ;
END_VAR
(************Ovládanie Komunikácie s tlačiarňou*******************)
VAR
	Client : Client_typ;
	Tlaciaren : Tlaciaren_typ;
	EtiketaPanasonic : EtiketaPanasonic_typ := (0);
END_VAR
(******************Blikače*****************************)
VAR
	Blikac100ms : BOOL;
	Blikac200ms : BOOL;
	Blikac500ms : BOOL;
	Blikac1s : BOOL;
END_VAR
(**************Remanentné premenné*********)
VAR
	RemPremenne : RemPremenne_typ;
	MpRecipeXml_0 : MpRecipeXml := (0);
	MpRecipeRegPar_0 : MpRecipeRegPar := (0);
	MpRecipeUI_0 : MpRecipeUI;
	UlozPremenne : BOOL;
	NacitajPremenne : BOOL;
END_VAR
VAR RETAIN
	VstupVytah_Banner_AKTIVNY : BOOL := FALSE;
	VystupVytah_Banner_AKTIVNY : BOOL := FALSE;
	VystupVytah_BannerNG_AKTIVNY : BOOL := FALSE;
END_VAR
(*************Premenne receptur**************)
VAR
	Receptura : ARRAY[0..150] OF ParametreRecepturTyp := [151((0))];
	MpRecipeXml_1 : MpRecipeXml := (0);
	MpRecipeRegPar_1 : MpRecipeRegPar := (0);
	ZoznamReceptur : ARRAY[0..150] OF STRING[50] := [151('')];
	UlozRecepturu : BOOL := FALSE;
	VymazRecepturu : BOOL := FALSE;
	NacitajRecepturu : BOOL;
	PrepisRecepturu : BOOL := FALSE;
	NazovModelu : STRING[18] := '';
	TypPaletky : STRING[10] := '';
	Robot_CisloProgramu : USINT;
	Kamera_CisloProgramu_QRkod : USINT := 0;
	Kamera_CisloProgramu_DMkod : USINT := 0;
	RychlostDopravnikaPriCisteni : REAL := 0.0;
	OffsetRobota_NazovModelu : STRING[18] := '';
	NacitajKorekcieRobota : BOOL := FALSE;
	UlozKorekcieRobota : BOOL := FALSE;
	UlozenieKorekcii_DONE : BOOL := FALSE;
	NacitanieKorekcii_DONE : BOOL := FALSE;
END_VAR
(***************Historia výroby*************************************)
VAR RETAIN
	HistoriaVyroby : ARRAY[0..5] OF HystoriaVyroby_typ := [6((0))];
	IndexHistorie : USINT := 0;
	Zvoleny_MODEL : STRING[18] := '';
	Zvoleny_LOT : STRING[11] := '';
END_VAR
(**********Premenne uzivatelov********************************)
VAR
	Uzivatel : ARRAY[0..50] OF ParametreUzivatelovTyp;
	MpRecipeXml_2 : MpRecipeXml := (0);
	MpRecipeRegPar_2 : MpRecipeRegPar := (0);
	ZoznamUzivatelov : ARRAY[0..50] OF STRING[50] := [51('')];
	MenoUzivatela : STRING[50];
	HesloUzivatela : STRING[50];
	UrovenUzivatela : UINT;
	ZadaneMenoUzivatela : STRING[50];
	ZadaneHesloUzivatela : STRING[50];
	ZvolenyUzivatel : STRING[50];
	ZvolenaUroven : UINT;
	TP_ZobrazPopUpPrihlasenie : USINT;
	UlozUzivatelov : BOOL;
	PrihlasUzivatela : BOOL;
	VymazUzivatela : BOOL;
	OdhlasUzivatela : BOOL;
	SC_Uzivatelia : SequenceControlTyp;
END_VAR
(*************Všeobecné premenné*************)
VAR
	Vizu : Vizu_typ;
	Safety : Safety_typ;
END_VAR
VAR RETAIN
	Paletka : ARRAY[0..200] OF Paletka_typ;
END_VAR
VAR
	StavHardware : Hardware_STAV_typ := (0);
	Kamera : CAM_typ := (0);
	Linka : Linka_typ := (0);
	VstupVytah : VstupnyVytah_typ := (0);
	SC_VstupVytah : SequenceControlTyp := (0);
	StoperPredCistenim : StoperPredCistenim_typ := (0);
	SC_StoperPredCistenim : SequenceControlTyp := (0);
	StoperPoCisteni : StoperPoCisteni_typ := (0);
	SC_StoperPoCisteni : SequenceControlTyp := (0);
	DopravCistenia : DopravCistenia_typ := (0);
	SC_DopravCistenia : SequenceControlTyp := (0);
	StoperEtiketovania : StoperEtiketovania_typ := (0);
	SC_StoperEtiketovania : SequenceControlTyp := (0);
	Robot : Robot_typ := (0);
	SC_Robot : SequenceControlTyp := (0);
	StoperDopravNG : StoperDopravnikaNG_typ := (0);
	SC_StoperDopravNG : SequenceControlTyp := (0);
	DopravBunky : DopravBunky_typ := (0);
	SC_DopravBunky : SequenceControlTyp := (0);
	StoperVystupDopravnika : StoperVystupDopravnika_typ := (0);
	SC_StoperVystupDopravnika : SequenceControlTyp := (0);
	VystupnyDopravnik : VystupnyDopravnik_typ := (0);
	SC_VystupnyDopravnik : SequenceControlTyp := (0);
	VystupVytah : VystupnyVytah_typ := (0);
	SC_VystupVytah : SequenceControlTyp := (0);
	StoperVratDopravnika : StoperVratDopravnika_typ := (0);
	SC_StoperVratDopravnika : SequenceControlTyp := (0);
	VratnyDopravnik : VratnyDopravnik_typ := (0);
	SC_VratnyDopravnik : SequenceControlTyp := (0);
END_VAR
(*****************Alarmy*****************************)
VAR
	Alarmy : ARRAY[0..100] OF BOOL;
	NastalaPorucha : BOOL;
	PotvrdenieAlarmov : BOOL;
	PoruchaLinky : BOOL := FALSE;
	PoruchaVstupnehoVytahu : BOOL;
	PoruchaCistenia : BOOL := FALSE;
	PoruchaBunky : BOOL;
	PoruchaVystupnehoVytahu : BOOL;
END_VAR
(***********Štatistiky pracovisk*******************)
VAR
	VstupnyVytah_Statistika : Taktime := (0);
	StoperPredCistenim_Statistika : Taktime := (0);
	StoperPoCisteni_Statistika : Taktime := (0);
	StoperEtiketovania_Statistika : Taktime := (0);
	StoperDopravNG_Statistika : Taktime := (0);
	VystupnyVytah_Statistika : Taktime := (0);
END_VAR
VAR RETAIN
	Linka_Statistika : Taktime := (0);
	PocetVyrobenychKusov_OK : REAL := 0.0;
	PocetVyrobenychKusov_NG : REAL := 0.0;
	CelkovyPocetVyrobenychKusov : UDINT := 0;
END_VAR
VAR
	Pomer_OK_kusov_IDR : REAL := 0.0;
	RESET_PoctuVyrobenychKusov : BOOL := FALSE;
	RESET_CelkovehoPoctuKusov : BOOL := FALSE;
END_VAR
(*************Motohodiny*************************)
VAR RETAIN
	Tajfun_Motohodiny : Motohodiny_typ := (0);
END_VAR
(************* Komunikacia Ethernet_IP ********************************)
VAR
	KOM_Panasonic : KOM_EthernetIP := (0);
END_VAR
```

### Package Logical/Libraries - Global libraries

### Library Logical/Libraries/FM_NORD (IEC)

#### Types.typ - Exported data types
```iecst
TYPE
	MenicSTAV_typ : 	STRUCT
		PORUCHA : BOOL;
		Pozicia_DOSIAHNUTA : BOOL;
		RUN : BOOL;
		READY : BOOL;
		Homing_OK : BOOL;
		ParamSada_BIT0_ENABLE : BOOL;
		ParamSada_BIT1_ENABLE : BOOL;
		QuickStop_Aktivny : BOOL;
		Komunikacia_OK : BOOL;
	END_STRUCT;
	MenicCMD_typ : 	STRUCT
		Chod_VPRED : BOOL;
		Chod_VZAD : BOOL;
		QuickSTOP : BOOL;
		Polohuj : BOOL;
		Potvrd_PORUCHU : BOOL;
		HOME : BOOL;
		Pozicia_RESET : BOOL;
	END_STRUCT;
	MenicPAR_typ : 	STRUCT
		ZadanaFrekvencia_Hz : REAL;
		AktualnaFrekvencia_Hz : REAL;
		AktualnyMoment_Nm : REAL;
		ZadanaPozicia_MM : UDINT;
		AktualnaPozicia_MM : UDINT;
		TypKomunikacieProfinet : BOOL; (*0 - Powerlink, 1- Profinet*)
		SwapovanieKomunikacie : BOOL; (*0 - NIE, 1 - ANO*)
		BUS_IN_Bit_0 : BOOL;
		BUS_IN_Bit_1 : BOOL;
		BUS_IN_Bit_2 : BOOL;
		BUS_IN_Bit_3 : BOOL;
		BUS_IN_Bit_4 : BOOL;
		BUS_IN_Bit_5 : BOOL;
		BUS_IN_Bit_6 : BOOL;
		BUS_OUT_Bit_0 : BOOL;
		BUS_OUT_Bit_1 : BOOL;
		BUS_OUT_Bit_2 : BOOL;
		BUS_OUT_Bit_3 : BOOL;
		BUS_OUT_Bit_4 : BOOL;
		BUS_OUT_Bit_5 : BOOL;
		BUS_OUT_Bit_6 : BOOL;
	END_STRUCT;
	PowerlinkKOM_IN_typ : 	STRUCT
		StavoveSlovo : UINT;
		StavovaHodnota_1 : INT;
		StavovaHodnota_2 : INT;
		StavovaHodnota_3 : INT;
		StavovaHodnota_4 : INT;
		StavovaHodnota_5 : INT;
	END_STRUCT;
	PowerlinkKOM_OUT_typ : 	STRUCT
		RiadiaceSlovo : UINT;
		ZadanaHodnota_1 : INT;
		ZadanaHodnota_2 : INT;
		ZadanaHodnota_3 : INT;
		ZadanaHodnota_4 : INT;
		ZadanaHodnota_5 : INT;
	END_STRUCT;
	ProfinetKOM_IN_typ : 	STRUCT
		StavoveSlovo : UINT;
		StavovaHodnota_1 : UINT;
		StavovaHodnota_2 : UINT;
		StavovaHodnota_3 : UINT;
		StavovaHodnota_4 : UINT;
		StavovaHodnota_5 : UINT;
	END_STRUCT;
	ProfinetKOM_OUT_typ : 	STRUCT
		RiadiaceSlovo : UINT;
		ZadanaHodnota_1 : UINT;
		ZadanaHodnota_2 : UINT;
		ZadanaHodnota_3 : UINT;
		ZadanaHodnota_4 : UINT;
		ZadanaHodnota_5 : UINT;
	END_STRUCT;
END_TYPE
```

#### FM_NORD.fun - Exported functions and function blocks
```iecst
{REDUND_ERROR} FUNCTION_BLOCK RiadenieFM (*Blok pre riadenie frekvencneho menica na Powerlinku*) (*$GROUP=User,$CAT=User,$GROUPICON=User.png,$CATICON=User.png*)
	VAR_INPUT
		CMD : MenicCMD_typ;
		PAR : MenicPAR_typ;
		Powerlink_KOM_IN : PowerlinkKOM_IN_typ;
		Profinet_KOM_IN : ProfinetKOM_IN_typ;
	END_VAR
	VAR_OUTPUT
		Powerlink_KOM_OUT : PowerlinkKOM_OUT_typ;
		Profinet_KOM_OUT : ProfinetKOM_OUT_typ;
		STAV : MenicSTAV_typ;
	END_VAR
	VAR
		Step : USINT;
		SCAL_ZadanejFrekvencie : LCRScal;
		SCAL_AktualnejFrekvencie : LCRScal;
		SCAL_AktualnehoMomentu : LCRScal;
		CONV_ZadPoz_UDINT_to_UINT : UdintToUint;
		CONV_AktPoz_UINT_to_UDINT : UintToUdint;
		ZadanaFrekvencia_preFM : INT;
		AktualnaFrekvencia_zFM_REAL : REAL;
		AktualnaFrekvencia_zFM : INT;
		AktualnyMoment_zFM : INT;
		AktualnyMoment_zFM_REAL : REAL;
		ZadanaPozicia_LW_preFM : INT;
		ZadanaPozicia_HW_preFM : INT;
		AktualnaPozicia_LW_zFM : INT;
		AktualnaPozicia_HW_zFM : INT;
		StavoveSlovo : UINT;
		StavovaHodnota_1 : UINT;
		StavovaHodnota_2 : UINT;
		StavovaHodnota_3 : UINT;
		StavovaHodnota_4 : UINT;
		StavovaHodnota_5 : UINT;
		RiadiaceSlovo : UINT;
		ZadanaHodnota_1 : UINT;
		ZadanaHodnota_2 : UINT;
		ZadanaHodnota_3 : UINT;
		ZadanaHodnota_4 : UINT;
		ZadanaHodnota_5 : UINT;
		zzEdge00000 : BOOL;
		CasHomingu : TON;
		CasPolohovania : TON;
	END_VAR
END_FUNCTION_BLOCK

{REDUND_ERROR} {REDUND_UNREPLICABLE} FUNCTION_BLOCK UintToUdint (*Prevod 16 bitových premenných do jednej 32 bitovej premennej*) (*$GROUP=User,$CAT=User,$GROUPICON=User.png,$CATICON=User.png*)
	VAR_INPUT
		InputArrayUINT : {REDUND_UNREPLICABLE} ARRAY[0..1] OF UINT;
	END_VAR
	VAR_OUTPUT
		OutputUDINT : {REDUND_UNREPLICABLE} UDINT;
	END_VAR
END_FUNCTION_BLOCK

{REDUND_ERROR} {REDUND_UNREPLICABLE} FUNCTION_BLOCK UdintToUint (*Prevod 32 bitovej premennej do 16 bitových premenných*) (*$GROUP=User,$CAT=User,$GROUPICON=User.png,$CATICON=User.png*)
	VAR_INPUT
		InputUDINT : {REDUND_UNREPLICABLE} UDINT;
	END_VAR
	VAR_OUTPUT
		OutputArrayUINT : {REDUND_UNREPLICABLE} ARRAY[0..1] OF UINT;
	END_VAR
END_FUNCTION_BLOCK
```

#### RiadenieFM.st
```iecst
(* Blok pre riadenie frekvencneho menica na Powerlinku *)
FUNCTION_BLOCK RiadenieFM

		//***********************************Control word************************************//
 	//Bit_0 - RUN
	//Bit_1 - Disable Voltage
	//Bit_2 - Quick Stop
	//Bit_3 - Enable Operation
	//Bit_4 - Pulse Enabled
	//Bit_5 - Enable Ramp
	//Bit_6 - Setpoint Enabled
	//Bit_7 - Potvrdenie poruchy
	//Bit_8 - Činnosť zadana v parametry maniča P480_11 /Homing Štart//
	//Bit_9 - Činnosť zadana v parametry meniča P480_12 /Reset pozície alebo referenčný bod/
	//Bit_10 - Zapnutie riadenie meniča cez komunikáciu
	//Bit_11 - Smer otáčania vpravo
	//Bit_12 - Smer otáčania vľavo
	//Bit_13 - Reserve
	//Bit_14 - Prepnutie parametrovej sady - bit 0
	//Bit_15 - Prepnutie parametrovej sady - bit 1

	//*************************************Status word*************************************//
	//Bit_0 - Stav READY
	//Bit_1 - READY for operation
	//Bit_2 - Stav motor beží
	//Bit_3 - Porucha
	//Bit_4 - Voltage Enabled
	//Bit_5 - Stav Quick Stop /0 - Quick stop aktívny, 1 - Quick stop neaktívny/
	//Bit_6 - No starting lockout
	//Bit_7 - Warning
	//Bit_8 - Pozícia dosiahnutá
	//Bit_9 - Bus control active
	//Bit_10 - Stav zadaný v parametri meniča P481_11 aktivny /Homing OK/
	//Bit_11 - Stav motor beží vpravo
	//Bit_12 - Stav motor beží vľavo
	//Bit_13 - Stav zadaný v parametri meniča P481_12 aktívny
	//Bit_14 - Stav prepnutia parametrovej sady - bit 0
	//Bit_15 - Stav prepnutia parametrovej sady - bit 1

	//***************************Prehodenie bitov komunikácie**********************************************//
	IF PAR.TypKomunikacieProfinet = 0 THEN //Powerlink//
		StavoveSlovo:= Powerlink_KOM_IN.StavoveSlovo;
		StavovaHodnota_1:= Powerlink_KOM_IN.StavovaHodnota_1;
		StavovaHodnota_2:= Powerlink_KOM_IN.StavovaHodnota_2;
		StavovaHodnota_3:= Powerlink_KOM_IN.StavovaHodnota_3;
		StavovaHodnota_4:= Powerlink_KOM_IN.StavovaHodnota_4;
		StavovaHodnota_5:= Powerlink_KOM_IN.StavovaHodnota_5;

		Powerlink_KOM_OUT.RiadiaceSlovo:= RiadiaceSlovo;
		Powerlink_KOM_OUT.ZadanaHodnota_1:= ZadanaHodnota_1;
		Powerlink_KOM_OUT.ZadanaHodnota_2:= ZadanaHodnota_2;
		Powerlink_KOM_OUT.ZadanaHodnota_3:= ZadanaHodnota_3;
		Powerlink_KOM_OUT.ZadanaHodnota_4:= ZadanaHodnota_4;
		Powerlink_KOM_OUT.ZadanaHodnota_5:= ZadanaHodnota_5;

	ELSIF PAR.TypKomunikacieProfinet = 1 THEN  //Profinet//
		IF PAR.SwapovanieKomunikacie = 0 THEN
			StavoveSlovo:= Profinet_KOM_IN.StavoveSlovo;
			StavovaHodnota_1:= Profinet_KOM_IN.StavovaHodnota_1;
			StavovaHodnota_2:= Profinet_KOM_IN.StavovaHodnota_2;
			StavovaHodnota_3:= Profinet_KOM_IN.StavovaHodnota_3;
			StavovaHodnota_4:= Profinet_KOM_IN.StavovaHodnota_4;
			StavovaHodnota_5:= Profinet_KOM_IN.StavovaHodnota_5;

			Profinet_KOM_OUT.RiadiaceSlovo:= RiadiaceSlovo;
			Profinet_KOM_OUT.ZadanaHodnota_1:= ZadanaHodnota_1;
			Profinet_KOM_OUT.ZadanaHodnota_2:= ZadanaHodnota_2;
			Profinet_KOM_OUT.ZadanaHodnota_3:= ZadanaHodnota_3;
			Profinet_KOM_OUT.ZadanaHodnota_4:= ZadanaHodnota_4;
			Profinet_KOM_OUT.ZadanaHodnota_5:= ZadanaHodnota_5;

		ELSIF PAR.SwapovanieKomunikacie = 1 THEN
			StavoveSlovo:= swapUINT(Profinet_KOM_IN.StavoveSlovo);
			StavovaHodnota_1:= swapUINT(Profinet_KOM_IN.StavovaHodnota_1);
			StavovaHodnota_2:= swapUINT(Profinet_KOM_IN.StavovaHodnota_2);
			StavovaHodnota_3:= swapUINT(Profinet_KOM_IN.StavovaHodnota_3);
			StavovaHodnota_4:= swapUINT(Profinet_KOM_IN.StavovaHodnota_4);
			StavovaHodnota_5:= swapUINT(Profinet_KOM_IN.StavovaHodnota_5);

			Profinet_KOM_OUT.RiadiaceSlovo:= swapUINT(RiadiaceSlovo);
			Profinet_KOM_OUT.ZadanaHodnota_1:= swapUINT(ZadanaHodnota_1);
			Profinet_KOM_OUT.ZadanaHodnota_2:= swapUINT(ZadanaHodnota_2);
			Profinet_KOM_OUT.ZadanaHodnota_3:= swapUINT(ZadanaHodnota_3);
			Profinet_KOM_OUT.ZadanaHodnota_4:= swapUINT(ZadanaHodnota_4);
			Profinet_KOM_OUT.ZadanaHodnota_5:= swapUINT(ZadanaHodnota_5);

		END_IF
	END_IF

	//***************************Preposielanie IO bitov**********************************************//
	//Vstupy pre menič//
	ZadanaHodnota_4.0:= PAR.BUS_IN_Bit_0;
	ZadanaHodnota_4.1:= PAR.BUS_IN_Bit_1;
	ZadanaHodnota_4.2:= PAR.BUS_IN_Bit_2;
	ZadanaHodnota_4.3:= PAR.BUS_IN_Bit_3;
	ZadanaHodnota_4.4:= PAR.BUS_IN_Bit_4;
	ZadanaHodnota_4.5:= PAR.BUS_IN_Bit_5;
	ZadanaHodnota_4.6:= PAR.BUS_IN_Bit_6;

	//Výstupy z meniča//
	PAR.BUS_OUT_Bit_0:= StavovaHodnota_4.0;
	PAR.BUS_OUT_Bit_1:= StavovaHodnota_4.1;
	PAR.BUS_OUT_Bit_2:= StavovaHodnota_4.2;
	PAR.BUS_OUT_Bit_3:= StavovaHodnota_4.3;
	PAR.BUS_OUT_Bit_4:= StavovaHodnota_4.4;
	PAR.BUS_OUT_Bit_5:= StavovaHodnota_4.5;
	PAR.BUS_OUT_Bit_6:= StavovaHodnota_4.6;

	//Zadaná frekvencia//
	ZadanaHodnota_1:= ZadanaFrekvencia_preFM;

	//Aktuálna frekvencia//
	AktualnaFrekvencia_zFM:= StavovaHodnota_1;
	//Zadaná pozícia//
	ZadanaHodnota_2:= ZadanaPozicia_LW_preFM;
	ZadanaHodnota_3:= ZadanaPozicia_HW_preFM;
	//Aktuálna pozícia//
	AktualnaPozicia_LW_zFM:= StavovaHodnota_2;
	AktualnaPozicia_HW_zFM:= StavovaHodnota_3;

	//***********************************************Stavy meniča******************************************************//
	STAV.PORUCHA:= StavoveSlovo.3;
	STAV.QuickStop_Aktivny:= NOT StavoveSlovo.5;
	STAV.READY:= StavoveSlovo.0;
	STAV.RUN:= StavoveSlovo.2;
	STAV.Pozicia_DOSIAHNUTA:= StavoveSlovo.8;
	STAV.Homing_OK:= StavoveSlovo.10;
	STAV.ParamSada_BIT0_ENABLE:= StavoveSlovo.14;
	STAV.ParamSada_BIT1_ENABLE:= StavoveSlovo.15;

	//Škálovanie zadanej frekvencie - Parameter meniča 105 = 50Hz//
	SCAL_ZadanejFrekvencie(x:= PAR.ZadanaFrekvencia_Hz, x1:= 0.0, y1:= 0.0, x2:= 50.0, y2:= 16384.0);
	ZadanaFrekvencia_preFM:= REAL_TO_INT(SCAL_ZadanejFrekvencie.y);

	//Škálovanie aktualnej frekvencie - Parameter meniča 105 = 50Hz//
	AktualnaFrekvencia_zFM_REAL:= INT_TO_REAL(AktualnaFrekvencia_zFM);
	SCAL_AktualnejFrekvencie(x:= AktualnaFrekvencia_zFM_REAL, x1:= 0.0, y1:= 0.0, x2:= 16384.0, y2:= 50.0);
	PAR.AktualnaFrekvencia_Hz:= SCAL_AktualnejFrekvencie.y;

	//Škálovanie aktuálneho momentu//
	AktualnyMoment_zFM_REAL:= INT_TO_REAL(AktualnyMoment_zFM);
	SCAL_AktualnehoMomentu(x:= AktualnyMoment_zFM_REAL, x1:= 0.0, y1:= 0.0, x2:= 16384.0, y2:= 100.0);
	PAR.AktualnyMoment_Nm:= SCAL_AktualnehoMomentu.y;

	//Rozloženie 32 bitovej hodnoty UDINT na dve 16 bitove hodnoty UINT pri zadávanie pozicie//
	CONV_ZadPoz_UDINT_to_UINT.InputUDINT:= PAR.ZadanaPozicia_MM;
	ZadanaPozicia_LW_preFM:= CONV_ZadPoz_UDINT_to_UINT.OutputArrayUINT[0];
	ZadanaPozicia_HW_preFM:= CONV_ZadPoz_UDINT_to_UINT.OutputArrayUINT[1];
	CONV_ZadPoz_UDINT_to_UINT();

	//Spojenie dvoch 16 bitových hodnot UINT do jednej 32 bitovej hodnoty UDINT pre čítanie pozicie//
	CONV_AktPoz_UINT_to_UDINT.InputArrayUINT[0]:= AktualnaPozicia_LW_zFM;
	CONV_AktPoz_UINT_to_UDINT.InputArrayUINT[1]:= AktualnaPozicia_HW_zFM;
	PAR.AktualnaPozicia_MM:= CONV_AktPoz_UINT_to_UDINT.OutputUDINT;
	CONV_AktPoz_UINT_to_UDINT();

	//Potvrdenie poruchy//
	IF CMD.Potvrd_PORUCHU THEN
		RiadiaceSlovo:= 16#4FE;
		IF NOT STAV.PORUCHA THEN
			RiadiaceSlovo:= 16#47E;
			CMD.Potvrd_PORUCHU:= FALSE;
		END_IF
	END_IF

	//Quick stop//
	IF CMD.QuickSTOP THEN
		Step:= 0;
		RiadiaceSlovo:= 16#47A;
		IF STAV.QuickStop_Aktivny THEN
			RiadiaceSlovo:= 16#47E;
			CMD.QuickSTOP:= FALSE;
		END_IF
	END_IF

	//Reset polohy meniča//
	IF CMD.Pozicia_RESET THEN
		RiadiaceSlovo:= 16#67E;
		IF PAR.AktualnaPozicia_MM = 0 THEN
			RiadiaceSlovo:= 16#47E;
			CMD.Pozicia_RESET:= FALSE;
		END_IF
	END_IF

	//Parametrové sady//
	//Bit_0 = 0,Bit_1 = 0 - Parametrova sada 1
	//Bit_0 = 1,Bit_1 = 0 - Parametrova sada 2 (Polohovanie)
	//Bit_0 = 0,Bit_1 = 1 - Parametrova sada 3
	//Bit_0 = 1,Bit_1 = 1 - Parametrova sada 4

	//Riadenie meniča//

	CASE Step OF

		0: //Nulovanie//
			CMD.HOME:= FALSE;
			CMD.Chod_VPRED:= FALSE;
			CMD.Chod_VZAD:= FALSE;
			CMD.Polohuj:= FALSE;
			CasHomingu.IN:= FALSE;
			CasPolohovania.IN:= FALSE;
			IF STAV.READY AND NOT STAV.PORUCHA AND NOT CMD.QuickSTOP THEN
				RiadiaceSlovo:= 16#47E;
				Step:= 1;
			END_IF

		1: //Rozhodnutie o činnosti//
			IF CMD.HOME THEN
				Step:= 10;
			ELSIF CMD.Chod_VPRED THEN
				Step:= 20;
			ELSIF CMD.Chod_VZAD THEN
				Step:= 30;
			ELSIF CMD.Polohuj THEN
				Step:= 40;
			END_IF

		10: //Štart homingu//
			IF PAR.ZadanaFrekvencia_Hz = 0.0 THEN
				PAR.ZadanaFrekvencia_Hz:= 5;
			END_IF

			RiadiaceSlovo:= 16#557F;
			CasHomingu.IN:= TRUE;
			Step:= 11;

		11: //Ukončenie homingu//
			IF STAV.Homing_OK AND CasHomingu.Q THEN
				RiadiaceSlovo:= 16#47E;
				Step:= 0;
			ELSIF NOT CMD.HOME THEN
				RiadiaceSlovo:= 16#47E;
				Step:= 0;
			END_IF

		20: //Chod VPRED//
			IF PAR.ZadanaFrekvencia_Hz = 0.0 THEN
				PAR.ZadanaFrekvencia_Hz:= 10;
			END_IF

			RiadiaceSlovo:= 16#C7F;

			IF NOT CMD.Chod_VPRED THEN
				RiadiaceSlovo:= 16#47E;
				Step:= 0;
			END_IF

		30: //Chod VZAD//
			IF PAR.ZadanaFrekvencia_Hz = 0.0 THEN
				PAR.ZadanaFrekvencia_Hz:= 10;
			END_IF

			RiadiaceSlovo:= 16#147F;

			IF NOT CMD.Chod_VZAD THEN
				RiadiaceSlovo:= 16#47E;
				Step:= 0;
			END_IF

		40: //Štart polohovania//
			IF PAR.ZadanaFrekvencia_Hz = 0.0 THEN
				PAR.ZadanaFrekvencia_Hz:= 10;
			END_IF

			IF PAR.AktualnaPozicia_MM <> PAR.ZadanaPozicia_MM THEN
				RiadiaceSlovo:= 16#447F;
				CasPolohovania.IN:= TRUE;
				Step:= 41;
			ELSE
				Step:= 0;
			END_IF

		41:	//Ukončenie polohovanie//

			IF STAV.Pozicia_DOSIAHNUTA AND CasPolohovania.Q THEN
				RiadiaceSlovo:= 16#47E;
				Step:= 0;
			ELSIF NOT CMD.Polohuj THEN
				RiadiaceSlovo:= 16#47E;
				Step:= 0;
			END_IF

	END_CASE

	CasHomingu.PT:= T#500ms;
	CasHomingu();

	CasPolohovania.PT:= T#500ms;
	CasPolohovania();

END_FUNCTION_BLOCK
```

#### UdintToUint.st
```iecst
(* TODO: Add your comment here *)
FUNCTION_BLOCK UdintToUint

	//Prevod UDINT do premenných UINT//
	OutputArrayUINT[0].0:= InputUDINT.0;
	OutputArrayUINT[0].1:= InputUDINT.1;
	OutputArrayUINT[0].2:= InputUDINT.2;
	OutputArrayUINT[0].3:= InputUDINT.3;
	OutputArrayUINT[0].4:= InputUDINT.4;
	OutputArrayUINT[0].5:= InputUDINT.5;
	OutputArrayUINT[0].6:= InputUDINT.6;
	OutputArrayUINT[0].7:= InputUDINT.7;
	OutputArrayUINT[0].8:= InputUDINT.8;
	OutputArrayUINT[0].9:= InputUDINT.9;
	OutputArrayUINT[0].10:= InputUDINT.10;
	OutputArrayUINT[0].11:= InputUDINT.11;
	OutputArrayUINT[0].12:= InputUDINT.12;
	OutputArrayUINT[0].13:= InputUDINT.13;
	OutputArrayUINT[0].14:= InputUDINT.14;
	OutputArrayUINT[0].15:= InputUDINT.15;
	OutputArrayUINT[1].0:= InputUDINT.16;
	OutputArrayUINT[1].1:= InputUDINT.17;
	OutputArrayUINT[1].2:= InputUDINT.18;
	OutputArrayUINT[1].3:= InputUDINT.19;
	OutputArrayUINT[1].4:= InputUDINT.20;
	OutputArrayUINT[1].5:= InputUDINT.21;
	OutputArrayUINT[1].6:= InputUDINT.22;
	OutputArrayUINT[1].7:= InputUDINT.23;
	OutputArrayUINT[1].8:= InputUDINT.24;
	OutputArrayUINT[1].9:= InputUDINT.25;
	OutputArrayUINT[1].10:= InputUDINT.26;
	OutputArrayUINT[1].11:= InputUDINT.27;
	OutputArrayUINT[1].12:= InputUDINT.28;
	OutputArrayUINT[1].13:= InputUDINT.29;
	OutputArrayUINT[1].14:= InputUDINT.30;
	OutputArrayUINT[1].15:= InputUDINT.31;

END_FUNCTION_BLOCK
```

#### UintToUdint.st
```iecst
(* TODO: Add your comment here *)
FUNCTION_BLOCK UintToUdint

	//Prevod UINT do premenné UDINT//
	OutputUDINT.0:= InputArrayUINT[0].0;
	OutputUDINT.1:= InputArrayUINT[0].1;
	OutputUDINT.2:= InputArrayUINT[0].2;
	OutputUDINT.3:= InputArrayUINT[0].3;
	OutputUDINT.4:= InputArrayUINT[0].4;
	OutputUDINT.5:= InputArrayUINT[0].5;
	OutputUDINT.6:= InputArrayUINT[0].6;
	OutputUDINT.7:= InputArrayUINT[0].7;
	OutputUDINT.8:= InputArrayUINT[0].8;
	OutputUDINT.9:= InputArrayUINT[0].9;
	OutputUDINT.10:= InputArrayUINT[0].10;
	OutputUDINT.11:= InputArrayUINT[0].11;
	OutputUDINT.12:= InputArrayUINT[0].12;
	OutputUDINT.13:= InputArrayUINT[0].13;
	OutputUDINT.14:= InputArrayUINT[0].14;
	OutputUDINT.15:= InputArrayUINT[0].15;
	OutputUDINT.16:= InputArrayUINT[1].0;
	OutputUDINT.17:= InputArrayUINT[1].1;
	OutputUDINT.18:= InputArrayUINT[1].2;
	OutputUDINT.19:= InputArrayUINT[1].3;
	OutputUDINT.20:= InputArrayUINT[1].4;
	OutputUDINT.21:= InputArrayUINT[1].5;
	OutputUDINT.22:= InputArrayUINT[1].6;
	OutputUDINT.23:= InputArrayUINT[1].7;
	OutputUDINT.24:= InputArrayUINT[1].8;
	OutputUDINT.25:= InputArrayUINT[1].9;
	OutputUDINT.26:= InputArrayUINT[1].10;
	OutputUDINT.27:= InputArrayUINT[1].11;
	OutputUDINT.28:= InputArrayUINT[1].12;
	OutputUDINT.29:= InputArrayUINT[1].13;
	OutputUDINT.30:= InputArrayUINT[1].14;
	OutputUDINT.31:= InputArrayUINT[1].15;

END_FUNCTION_BLOCK
```

### Library Logical/Libraries/SC (IEC)

#### Types.typ - Exported data types
```iecst
TYPE
	SequenceControlTyp : 	STRUCT
		StepName : STRING[200];
		Step : UINT;
		Switch1 : BOOL;
		Switch2 : BOOL;
		Switch3 : BOOL;
		ResetStep : BOOL;
		LastStep : BOOL;
		IdleTime : TON;
		AlarmTime : TON;
	END_STRUCT;
END_TYPE
```

#### SC.fun - Exported functions and function blocks
```iecst
FUNCTION SequenceControl : BOOL
	VAR_IN_OUT
		SC : SequenceControlTyp;
	END_VAR
END_FUNCTION
```

#### SequenceControl.st
```iecst
(* TODO: Add your comment here *)
FUNCTION SequenceControl

	IF SC.ResetStep THEN
		brsmemset(ADR(SC.StepName),0,SIZEOF(SC.StepName));
		SC.Switch1:= FALSE;
		SC.Switch2:= FALSE;
		SC.Switch3:= FALSE;
		SC.IdleTime.IN:= FALSE;
		SC.AlarmTime.IN:= FALSE;
		SC.ResetStep:= FALSE;
	END_IF

	IF SC.LastStep THEN
		brsmemset(ADR(SC.StepName),0,SIZEOF(SC.StepName));
		SC.Switch1:= FALSE;
		SC.Switch2:= FALSE;
		SC.Switch3:= FALSE;
		SC.IdleTime.IN:= FALSE;
		SC.AlarmTime.IN:= FALSE;
		SC.Step:= 0;
		SC.LastStep:= FALSE;
	END_IF

	//Volanie časovačov//
	SC.AlarmTime();
	SC.IdleTime();

END_FUNCTION
```

### Library Logical/Libraries/Statistika (IEC)

#### Types.typ - Exported data types
```iecst
TYPE
	Statistika_IN_typ : 	STRUCT
		START_MeraniaCasu : BOOL;
		ZAPIS_MeraniaCasu : BOOL;
		TaskovaTrieda_ms : UINT;
		RESET_CelkovehoCasu : BOOL;
		RESET_HistorieMeraniCasu : BOOL;
		RESET_PoctuKusov : BOOL;
		RESET_CelkovehoPoctuKusov : BOOL;
		PriratajKus_OK : BOOL;
		PriratajKus_NG : BOOL;
	END_STRUCT;
	Statistika_OUT_typ : 	STRUCT
		NameranyCas_v_Sekundach : REAL;
		NameranyCas_v_Minutach : REAL;
		NameranyCas_v_Hodinach : REAL;
		PriemernyCas_v_Sekundach : REAL;
		PriemernyCas_v_Minutach : REAL;
		Stav_ZapisCasu_DONE : BOOL;
		Stav_RESET_CelkCasu_DONE : BOOL;
		Stav_RESET_HistorieMerani_DONE : BOOL;
		HistoriaMerani_v_Sekundach : ARRAY[0..14]OF REAL;
		HistoriaMerani_v_Minutach : ARRAY[0..14]OF REAL;
		HistoriaMerani_v_Hodinach : ARRAY[0..14]OF REAL;
		CelkovyPocetNameranychSekund : REAL;
		CelkovyPocetNameranychMinut : REAL;
		CelkovyPocetNameranychHodin : REAL;
		Stav_PriratanieKusu_OK_DONE : BOOL;
		Stav_PriratanieKusu_NG_DONE : BOOL;
		PocetKusov_OK : UDINT;
		PocetKusov_NG : UDINT;
		CelkovyPocetKusov : UDINT;
		Stav_RESET_PoctuKusov_DONE : BOOL;
		Stav_RESET_CelkPoctuKusov_DONE : BOOL;
	END_STRUCT;
	Statistika_VAR_typ : 	STRUCT
		NameraneMilisekundy_REAL : REAL;
		NameraneSekundy_REAL : REAL;
		NameraneMinuty_REAL : REAL;
		NameraneHodiny_REAL : REAL;
		Milisekundy : UINT;
		Sekundy : UINT;
		Minuty : UINT;
		Hodiny : UINT;
		CelkoveSekundy : UINT;
		CelkoveMinuty : UINT;
		CelkoveHodiny : UINT;
		i : USINT;
		a : USINT;
		b : USINT;
		c : USINT;
		d : USINT;
		Priemer_SucetSekund_REAL : REAL;
		Priemer_SucetMinut_REAL : REAL;
		Priemer_SucetHodin_REAL : REAL;
	END_STRUCT;
END_TYPE
```

#### Statistika.fun - Exported functions and function blocks
```iecst
{REDUND_ERROR} FUNCTION_BLOCK Taktime (*Meranie taktime*) (*$GROUP=User,$CAT=User,$GROUPICON=User.png,$CATICON=User.png*)
	VAR_INPUT
		IN : Statistika_IN_typ;
	END_VAR
	VAR_OUTPUT
		OUT : Statistika_OUT_typ;
	END_VAR
	VAR
		IntVAR : Statistika_VAR_typ;
	END_VAR
END_FUNCTION_BLOCK
```

#### Taktime.st
```iecst
(* Meranie taktime *)
FUNCTION_BLOCK Taktime

//*********************************************************************Meranie taktime**************************************************************************//

    //Vynulovanie časovača//
	IF NOT IN.START_MeraniaCasu THEN
		IntVAR.Milisekundy:= 0;
		IntVAR.Sekundy:= 0;
		IntVAR.Minuty:= 0;
		IntVAR.Hodiny:= 0;
		IntVAR.CelkoveSekundy:= 0;
		IntVAR.CelkoveMinuty:= 0;
		IntVAR.CelkoveHodiny:= 0;
	END_IF

	//Zapnutie časovača//
	IF IN.START_MeraniaCasu THEN

		IntVAR.Milisekundy:= IntVAR.Milisekundy + IN.TaskovaTrieda_ms;//Ak je v taskovej triede 2ms tak prirátaváme + 2//

		IF IntVAR.Milisekundy >= 1000 THEN
			IntVAR.Sekundy:= IntVAR.Sekundy + 1;
			IntVAR.CelkoveSekundy:= IntVAR.CelkoveSekundy + 1;
			IntVAR.Milisekundy:= 0;
		END_IF

		IF IntVAR.Sekundy >= 60 THEN
			IntVAR.Minuty:= IntVAR.Minuty + 1;
			IntVAR.CelkoveMinuty:= IntVAR.CelkoveMinuty + 1;
			IntVAR.Sekundy:= 0;
		END_IF

		IF IntVAR.Minuty >= 60 THEN
			IntVAR.Hodiny:= IntVAR.Hodiny + 1;
			IntVAR.CelkoveHodiny:= IntVAR.CelkoveHodiny + 1;
			IntVAR.Minuty:= 0;
		END_IF

	END_IF

	//Ulozenie nameraného času a resetovanie časovača//
	IF IN.ZAPIS_MeraniaCasu AND NOT OUT.Stav_ZapisCasu_DONE THEN
		IntVAR.NameraneHodiny_REAL:= UINT_TO_REAL(IntVAR.CelkoveHodiny);
		IntVAR.NameraneMinuty_REAL:= UINT_TO_REAL(IntVAR.CelkoveMinuty);
		IntVAR.NameraneSekundy_REAL:= UINT_TO_REAL(IntVAR.CelkoveSekundy);
		IntVAR.NameraneMilisekundy_REAL:= UINT_TO_REAL(IntVAR.Milisekundy);
		//Zobrazenie celkového času v sekundách//
		OUT.NameranyCas_v_Sekundach:= IntVAR.NameraneSekundy_REAL + (IntVAR.NameraneMilisekundy_REAL / 1000);
		//Zobrazenie celkového času v minútach//
		OUT.NameranyCas_v_Minutach:= IntVAR.NameraneMinuty_REAL + (IntVAR.NameraneSekundy_REAL / 100);
		//Zobrazenie celkového času v hodinách//
		OUT.NameranyCas_v_Hodinach:= IntVAR.NameraneHodiny_REAL + (IntVAR.NameraneMinuty_REAL / 100);
		//Zápis do historie meraní//
		OUT.HistoriaMerani_v_Sekundach[IntVAR.i]:= OUT.NameranyCas_v_Sekundach;
		OUT.HistoriaMerani_v_Minutach[IntVAR.i]:= OUT.NameranyCas_v_Minutach;
		IntVAR.i:= IntVAR.i + 1;
		IF IntVAR.i > 14 THEN
			IntVAR.i:= 0;
		END_IF
		OUT.CelkovyPocetNameranychSekund:= OUT.CelkovyPocetNameranychSekund + OUT.NameranyCas_v_Sekundach;
		OUT.CelkovyPocetNameranychMinut:= OUT.CelkovyPocetNameranychMinut + OUT.NameranyCas_v_Minutach;
		OUT.CelkovyPocetNameranychHodin:= OUT.CelkovyPocetNameranychHodin + OUT.NameranyCas_v_Hodinach;
		IntVAR.Milisekundy:= 0;
		IntVAR.Sekundy:= 0;
		IntVAR.Minuty:= 0;
		IntVAR.Hodiny:= 0;
		IntVAR.CelkoveSekundy:= 0;
		IntVAR.CelkoveMinuty:= 0;
		IntVAR.CelkoveHodiny:= 0;
		OUT.Stav_ZapisCasu_DONE:= TRUE;
	END_IF

	IF NOT IN.ZAPIS_MeraniaCasu THEN
		OUT.Stav_ZapisCasu_DONE:= FALSE;
	END_IF

	//Vyrátanie priemernej hodnoty v sekundách//
	IntVAR.a:= 0;
	IntVAR.b:= 0;
	IntVAR.Priemer_SucetSekund_REAL:= 0;
	OUT.PriemernyCas_v_Sekundach:= 0;
	FOR IntVAR.a:= 0 TO 14 BY 1 DO
		IntVAR.Priemer_SucetSekund_REAL:= IntVAR.Priemer_SucetSekund_REAL + OUT.HistoriaMerani_v_Sekundach[IntVAR.a];
		IF OUT.HistoriaMerani_v_Sekundach[IntVAR.a] <> 0 THEN
			IntVAR.b:= IntVAR.b + 1;
		END_IF
		IF IntVAR.b <> 0 THEN
			OUT.PriemernyCas_v_Sekundach:= IntVAR.Priemer_SucetSekund_REAL / IntVAR.b;
		ELSE
			OUT.PriemernyCas_v_Sekundach:= 0;
		END_IF
	END_FOR

	//Vyrátanie priemernej hodnoty v minutách//
	IntVAR.c:= 0;
	IntVAR.d:= 0;
	IntVAR.Priemer_SucetMinut_REAL:= 0;
	OUT.PriemernyCas_v_Minutach:= 0;
	FOR IntVAR.c:= 0 TO 14 BY 1 DO
		IntVAR.Priemer_SucetMinut_REAL:= IntVAR.Priemer_SucetMinut_REAL + OUT.HistoriaMerani_v_Minutach[IntVAR.c];
		IF OUT.HistoriaMerani_v_Minutach[IntVAR.c] <> 0 THEN
			IntVAR.d:= IntVAR.d + 1;
		END_IF
		IF IntVAR.d <> 0 THEN
			OUT.PriemernyCas_v_Minutach:= IntVAR.Priemer_SucetMinut_REAL / IntVAR.d;
		ELSE
			OUT.PriemernyCas_v_Minutach:= 0;
		END_IF
	END_FOR

	//Reset celkových počítadiel času//
	IF IN.RESET_CelkovehoCasu AND NOT OUT.Stav_RESET_CelkCasu_DONE THEN
		OUT.CelkovyPocetNameranychSekund:= 0;
		OUT.CelkovyPocetNameranychMinut:= 0;
		OUT.CelkovyPocetNameranychHodin:= 0;
		OUT.Stav_RESET_CelkCasu_DONE:= TRUE;
	END_IF

	IF NOT IN.RESET_CelkovehoCasu THEN
		OUT.Stav_RESET_CelkCasu_DONE:= FALSE;
	END_IF

	//Reset historie merani//
	IF IN.RESET_HistorieMeraniCasu AND NOT OUT.Stav_RESET_HistorieMerani_DONE THEN
		brsmemset(ADR(OUT.HistoriaMerani_v_Sekundach),0,SIZEOF(OUT.HistoriaMerani_v_Sekundach));
		brsmemset(ADR(OUT.HistoriaMerani_v_Minutach),0,SIZEOF(OUT.HistoriaMerani_v_Minutach));
		OUT.Stav_RESET_HistorieMerani_DONE:= TRUE;
	END_IF

	IF NOT IN.RESET_HistorieMeraniCasu THEN
		OUT.Stav_RESET_HistorieMerani_DONE:= FALSE;
	END_IF

	//***************************************************************************Rátanie kusov****************************************************************************//

	//Rátanie kusov OK//
	IF IN.PriratajKus_OK AND NOT OUT.Stav_PriratanieKusu_OK_DONE THEN
		OUT.CelkovyPocetKusov:= OUT.CelkovyPocetKusov + 1;
		OUT.PocetKusov_OK:= OUT.PocetKusov_OK + 1;
		OUT.Stav_PriratanieKusu_OK_DONE:= TRUE;
	END_IF

	IF NOT IN.PriratajKus_OK THEN
		OUT.Stav_PriratanieKusu_OK_DONE:= FALSE;
	END_IF

	//Rátanie kusov NG//
	IF IN.PriratajKus_NG AND NOT OUT.Stav_PriratanieKusu_NG_DONE THEN
		OUT.CelkovyPocetKusov:= OUT.CelkovyPocetKusov + 1;
		OUT.PocetKusov_NG:= OUT.PocetKusov_NG + 1;
		OUT.Stav_PriratanieKusu_NG_DONE:= TRUE;
	END_IF

	IF NOT IN.PriratajKus_NG THEN
		OUT.Stav_PriratanieKusu_NG_DONE:= FALSE;
	END_IF

	//Reset počtu kusov //
	IF IN.RESET_PoctuKusov AND NOT OUT.Stav_RESET_PoctuKusov_DONE THEN
		OUT.PocetKusov_OK:= 0;
		OUT.PocetKusov_NG:= 0;
		OUT.Stav_RESET_PoctuKusov_DONE:= TRUE;
	END_IF

	IF NOT IN.RESET_PoctuKusov THEN
		OUT.Stav_RESET_PoctuKusov_DONE:= FALSE;
	END_IF

	//Reset celkového počtu kusov//
	IF IN.RESET_CelkovehoPoctuKusov AND NOT OUT.Stav_RESET_CelkPoctuKusov_DONE THEN
		OUT.CelkovyPocetKusov:= 0;
		OUT.Stav_RESET_CelkPoctuKusov_DONE:= TRUE;
	END_IF

	IF NOT IN.RESET_CelkovehoPoctuKusov THEN
		OUT.Stav_RESET_CelkPoctuKusov_DONE:= FALSE;
	END_IF

END_FUNCTION_BLOCK
```

### Library Logical/Libraries/IecCheck (IEC)
Depends on: sys_lib, AsBrStr

#### IecCheck.fun - Exported functions and function blocks
```iecst
FUNCTION CheckDivSint : SINT (* Check divisor for SINT division *)
	VAR_INPUT
		divisor : SINT;
	END_VAR
END_FUNCTION

FUNCTION CheckDivUsint : USINT (* Check divisor for USINT division *)
	VAR_INPUT
		divisor : USINT;
	END_VAR
END_FUNCTION

FUNCTION CheckDivInt : INT (* Check divisor for INT division *)
	VAR_INPUT
		divisor : INT;
	END_VAR
END_FUNCTION

FUNCTION CheckDivUint : UINT (* Check divisor for UINT division *)
	VAR_INPUT
		divisor : UINT;
	END_VAR
END_FUNCTION

FUNCTION CheckDivDint : DINT (* Check divisor for DINT division *)
	VAR_INPUT
		divisor : DINT;
	END_VAR
END_FUNCTION

FUNCTION CheckDivUdint : UDINT (* Check divisor for UDINT division *)
	VAR_INPUT
		divisor : UDINT;
	END_VAR
END_FUNCTION

FUNCTION CheckDivReal : REAL (* Check divisor for REAL division *)
	VAR_INPUT
		divisor : REAL;
	END_VAR
END_FUNCTION

FUNCTION CheckDivLReal : LREAL (* Check divisor for LREAL division, not available for SG3 and SGC *)
	VAR_INPUT
		divisor : LREAL;
	END_VAR
END_FUNCTION

FUNCTION CheckBounds : DINT (* Check range for array access *)
	VAR_INPUT
		index : DINT;
		lower : DINT;
		upper : DINT;
	END_VAR
END_FUNCTION

FUNCTION CheckRange : DINT (* Check range for enumeration *)
	VAR_INPUT
		value : DINT;
		lower : DINT;
		upper : DINT;
	END_VAR
END_FUNCTION

FUNCTION CheckSignedSubrange : DINT (* Check range for subrange of signed data types *)
	VAR_INPUT
		value : DINT;
		lower : DINT;
		upper : DINT;
	END_VAR
END_FUNCTION

FUNCTION CheckUnsignedSubrange : UDINT (* Check range for subrange of unsigned data types *)
	VAR_INPUT
		value : UDINT;
		lower : UDINT;
		upper : UDINT;
	END_VAR
END_FUNCTION

FUNCTION CheckReadAccess : UDINT (* Check address when reading dynamic variables *)
	VAR_INPUT
		address : UDINT;
	END_VAR
END_FUNCTION

FUNCTION CheckWriteAccess : UDINT (* Check address when writing dynamic variables *)
	VAR_INPUT
		address : UDINT;
	END_VAR
END_FUNCTION

FUNCTION MakeEntry : UDINT (* Makes an entry (log book entry) in the error log book *)
	VAR
		taskname : STRING[30];
		group : USINT;
		status_name : UINT;
		out_text : STRING[80];
	END_VAR
	VAR_INPUT
		number : UINT;
		index : DINT;
		text : STRING[50];
	END_VAR
END_FUNCTION
```

#### IecCheck.st - Implementation file
```iecst
(* Check divisor for SINT division *)
FUNCTION CheckDivSint
	IF divisor=0 THEN
		CheckDivSint:=1;
		MakeEntry(55555,divisor,'CheckDivSint');
	ELSE
		CheckDivSint:=divisor;
	END_IF
END_FUNCTION

(* Check divisor for USINT division *)
FUNCTION CheckDivUsint
	IF divisor=0 THEN
		CheckDivUsint:=1;
		MakeEntry(55555,divisor,'CheckDivUsint');
	ELSE
		CheckDivUsint:=divisor;
	END_IF
END_FUNCTION

(* Check divisor for INT division *)
FUNCTION CheckDivInt
	IF divisor=0 THEN
		CheckDivInt:=1;
		MakeEntry(55555,divisor,'CheckDivInt');
	ELSE
		CheckDivInt:=divisor;
	END_IF
END_FUNCTION

(* Check divisor for UINT division *)
FUNCTION CheckDivUint
	IF divisor=0 THEN
		CheckDivUint:=1;
		MakeEntry(55555,divisor,'CheckDivUint');
	ELSE
		CheckDivUint:=divisor;
	END_IF
END_FUNCTION

(* Check divisor for DINT division *)
FUNCTION CheckDivDint
	IF divisor=0 THEN
		CheckDivDint:=1;
		MakeEntry(55555,divisor,'CheckDivDint');
	ELSE
		CheckDivDint:=divisor;
	END_IF
END_FUNCTION

(* Check divisor for UDINT division *)
FUNCTION CheckDivUdint
	IF divisor=0 THEN
		CheckDivUdint:=1;
		MakeEntry(55555,divisor,'CheckDivUdint');
	ELSE
		CheckDivUdint:=divisor;
	END_IF
END_FUNCTION

(* Check divisor for REAL division *)
FUNCTION CheckDivReal
	IF divisor=0 THEN
		CheckDivReal:=1;
		MakeEntry(55555,0,'CheckDivReal');
	ELSE
		CheckDivReal:=divisor;
	END_IF
END_FUNCTION

(* Check divisor for LREAL division *)
FUNCTION CheckDivLReal
	IF divisor=0 THEN
		CheckDivLReal:=1;
		MakeEntry(55555,0,'CheckDivLReal');
	ELSE
		CheckDivLReal:=divisor;
	END_IF
END_FUNCTION

(* Check range for array access *)
FUNCTION CheckBounds
	IF index < lower THEN
		CheckBounds := lower;
		MakeEntry(55555,index,'CheckBounds');
	ELSIF index > upper THEN
		CheckBounds := upper;
		MakeEntry(55555,index,'CheckBounds');
	ELSE
		CheckBounds := index;
	END_IF
END_FUNCTION

(* Check range for enumeration *)
FUNCTION CheckRange
	IF value < lower THEN
		CheckRange := lower;
		MakeEntry(55555,value,'CheckRange');
	ELSIF value > upper THEN
		CheckRange := upper;
		MakeEntry(55555,value,'CheckRange');
	ELSE
		CheckRange := value;
	END_IF
END_FUNCTION

(* Check range for subrange of signed data types *)
FUNCTION CheckSignedSubrange
	IF value < lower THEN
		CheckSignedSubrange := lower;
		MakeEntry(55555,value,'CheckSignedSubrange');
	ELSIF value > upper THEN
		CheckSignedSubrange := upper;
		MakeEntry(55555,value,'CheckSignedSubrange');
	ELSE
		CheckSignedSubrange := value;
	END_IF
END_FUNCTION

(* Check range for subrange of unsigned data types *)
FUNCTION CheckUnsignedSubrange
	IF value < lower THEN
		CheckUnsignedSubrange := lower;
		MakeEntry(55555,value,'CheckUnsignedSubrange');
	ELSIF value > upper THEN
		CheckUnsignedSubrange := upper;
		MakeEntry(55555,value,'CheckUnsignedSubrange');
	ELSE
		CheckUnsignedSubrange := value;
	END_IF
END_FUNCTION

(* Check address when reading dynamic variables *)
FUNCTION CheckReadAccess
	IF address=0 THEN
		(* TODO: Insert an appropriate code, see AutomationStudio help for further information *)
		MakeEntry(55555,address,'Read from NULL');
	END_IF

	CheckReadAccess:=0;
END_FUNCTION

(* Check address when writing dynamic variables *)
FUNCTION CheckWriteAccess
	IF address=0 THEN
		(* TODO: Insert an appropriate code, see AutomationStudio help for further information *)
		MakeEntry(55555,address,'Write to NULL');
	END_IF

	CheckWriteAccess:=0;
END_FUNCTION

(* Makes an entry (log book entry) in the error log book *)
FUNCTION MakeEntry
		status_name := ST_name(0,ADR(taskname),ADR(group));

		brsstrcpy(ADR(out_text),ADR(text));
		brsstrcat(ADR(out_text),ADR(' > in task > '));
  		brsstrcat(ADR(out_text),ADR(taskname));
		MakeEntry := ADR(out_text);
		ERRxfatal(number,index,ADR(out_text));
END_FUNCTION
```

### Library Logical/Libraries/EthernetIP (IEC)

#### Types.typ - Exported data types
```iecst
TYPE
	Inputs_typ : 	STRUCT
		ProcessResult : BOOL;
		RFID_Reading_Error : BOOL;
		Blowing_Error : BOOL;
		QRcode_Reading_Error : BOOL;
		DMcode_Reading_Error : BOOL;
		Text_Reading_Error : BOOL;
		VytlacEtiketu_RucnyRezim : BOOL;
		RezimBezTlaceEtikety : BOOL;
		CommandNumber : UDINT;
		SerialNumber_InternaEtiketa : STRING[48];
		NazovPaletky_RFID : STRING[10];
		Cislo_LOTU : STRING[20];
		DataForServer_READY : BOOL;
	END_STRUCT;
	Outputs_typ : 	STRUCT
		ContinueToNextProcess : BOOL;
		SerialNumber_ZakaznickaEtiketa : STRING[49];
		ReturnProcessName : STRING[30];
		DataForPLC_READY : BOOL;
		LastCommandNumber : UDINT;
	END_STRUCT;
END_TYPE
```

#### EthernetIP.fun - Exported functions and function blocks
```iecst
{REDUND_ERROR} FUNCTION_BLOCK KOM_EthernetIP (*Komunikacia z Panasonic*) (*$GROUP=User,$CAT=User,$GROUPICON=User.png,$CATICON=User.png*)
	VAR_INPUT
		Server_IN : Inputs_typ;
		Mapping_IN : ARRAY[0..99] OF UDINT;
	END_VAR
	VAR_OUTPUT
		Server_OUT : Outputs_typ;
		Mapping_OUT : ARRAY[0..99] OF UDINT;
	END_VAR
	VAR
		SerNumber_InterEtiketa_PoleUSINT : ARRAY[0..47] OF USINT;
		SerNumber_InterEtiketa_PoleUDINT : ARRAY[0..47] OF UDINT;
		NazovPaletky_RFID_PoleUSINT : ARRAY[0..9] OF USINT;
		NazovPaletky_RFID_PoleUDINT : ARRAY[0..9] OF UDINT;
		Cislo_LOTU_PoleUSINT : ARRAY[0..19] OF USINT;
		Cislo_LOTU_PoleUDINT : ARRAY[0..19] OF UDINT;
		SerNumber_ZakazEtiketa_PoleUSINT : ARRAY[0..48] OF USINT;
		SerNumber_ZakazEtiketa_PoleUDINT : ARRAY[0..48] OF UDINT;
		ReturnProcessName_PoleUSINT : ARRAY[0..29] OF USINT;
		ReturnProcessName_PoleUDINT : ARRAY[0..29] OF UDINT;
		a : USINT;
		b : USINT;
		c : USINT;
		d : USINT;
		e : USINT;
	END_VAR
END_FUNCTION_BLOCK
```

#### KOM_EthernetIP.st
```iecst
(* Komunikacia z Panasonic *)
FUNCTION_BLOCK KOM_EthernetIP

	//**********************************Výstupy z PLC do Panasonic*******************************************************//
	//Výsledok procesu//
	Mapping_OUT[0].0:= Server_IN.ProcessResult;

	//Chyba čítania čipu paletky//
	Mapping_OUT[0].1:= Server_IN.RFID_Reading_Error;

	//Chyba v procese čistenia//
	Mapping_OUT[0].2:= Server_IN.Blowing_Error;

	//Chyba prečítania QR kódu interného štítku//
	Mapping_OUT[0].3:= Server_IN.QRcode_Reading_Error;

	//Chyba prečítania DM kódu zákaznickej etikety//
	Mapping_OUT[0].4:= Server_IN.DMcode_Reading_Error;

	//Chyba prečítania textu na zákaznickej etikete//
	Mapping_OUT[0].5:= Server_IN.Text_Reading_Error;

	//Vytlačenie etikety v ručnom režime//
	Mapping_OUT[0].6:= Server_IN.VytlacEtiketu_RucnyRezim;

	//Režim bez tlače etikety//
	Mapping_OUT[0].7:= Server_IN.RezimBezTlaceEtikety;

	//Číslo výrobného procesu//
	Mapping_OUT[1]:= Server_IN.CommandNumber;

	//Sériové číslo internej etikety//
	brsstrcpy(ADR(SerNumber_InterEtiketa_PoleUSINT),ADR(Server_IN.SerialNumber_InternaEtiketa));

	FOR a:= 0 TO 47 BY 1 DO
		SerNumber_InterEtiketa_PoleUDINT[a]:= SerNumber_InterEtiketa_PoleUSINT[a];
	END_FOR

	brsmemcpy(ADR(Mapping_OUT[2]),ADR(SerNumber_InterEtiketa_PoleUDINT),SIZEOF(SerNumber_InterEtiketa_PoleUDINT));

	//Názov paletky//
	brsstrcpy(ADR(NazovPaletky_RFID_PoleUSINT),ADR(Server_IN.NazovPaletky_RFID));

	FOR b:= 0 TO 9 BY 1 DO
		NazovPaletky_RFID_PoleUDINT[b]:= NazovPaletky_RFID_PoleUSINT[b];
	END_FOR

	brsmemcpy(ADR(Mapping_OUT[50]),ADR(NazovPaletky_RFID_PoleUDINT),SIZEOF(NazovPaletky_RFID_PoleUDINT));

	//Číslo LOTU//
	brsstrcpy(ADR(Cislo_LOTU_PoleUSINT),ADR(Server_IN.Cislo_LOTU));

	FOR c:= 0 TO 19 BY 1 DO
		Cislo_LOTU_PoleUDINT[c]:= Cislo_LOTU_PoleUSINT[c];
	END_FOR

	brsmemcpy(ADR(Mapping_OUT[60]),ADR(Cislo_LOTU_PoleUDINT),SIZEOF(Cislo_LOTU_PoleUDINT));

	//Potvrdenie dáta pre Panasonic pripravené//
	Mapping_OUT[80].0:= Server_IN.DataForServer_READY;

	//*********************************Vstupy z Panasonic do PLC*********************************************************//
	//Pokračovanie na další proces//
	Server_OUT.ContinueToNextProcess:= Mapping_IN[0].0;

	//Sériové číslo zákaznickej etikety//
	brsmemcpy(ADR(SerNumber_ZakazEtiketa_PoleUDINT),ADR(Mapping_IN[1]),196);

	FOR d:= 0 TO 48 BY 1 DO
		SerNumber_ZakazEtiketa_PoleUSINT[d]:= UDINT_TO_USINT(SerNumber_ZakazEtiketa_PoleUDINT[d]);
	END_FOR

	brsstrcpy(ADR(Server_OUT.SerialNumber_ZakaznickaEtiketa),ADR(SerNumber_ZakazEtiketa_PoleUSINT));

	//Return process name//
	brsmemcpy(ADR(ReturnProcessName_PoleUDINT),ADR(Mapping_IN[50]),120);

	FOR e:= 0 TO 29 BY 1 DO
		ReturnProcessName_PoleUSINT[e]:= UDINT_TO_USINT(ReturnProcessName_PoleUDINT[e]);
	END_FOR

	brsstrcpy(ADR(Server_OUT.ReturnProcessName),ADR(ReturnProcessName_PoleUSINT));

	//Potvrdenie dáta pre PLC pripravené//
	Server_OUT.DataForPLC_READY:= Mapping_IN[80].0;

	//Posledné prijaté číslo procesu//
	Server_OUT.LastCommandNumber:= Mapping_IN[81];

END_FUNCTION_BLOCK
```

### Package Logical/Program - Riadiace programy

### Program Logical/Program/Main (IEC)

#### Main.st - Init, cyclic, exit code
```iecst
PROGRAM _INIT

	Linka.CitackaQRkodu_AKTIVNA:= TRUE;

END_PROGRAM

PROGRAM _CYCLIC

	//Zapnutie osvetlenia bunky//
	IF NOT Linka.IN.PredneDvereZavrete_EZ1 OR NOT Linka.IN.ZadneDvereZavrete_EZ2 THEN
		Linka.OUT.OsvetlenieBunky_Zapni:= TRUE;
	ELSE
		Linka.OUT.OsvetlenieBunky_Zapni:= FALSE;
	END_IF

	//Ovládanie vzduchotechniky//
	IF Linka.OUT.IonJednotka_START THEN
		Linka.OUT.Vzduchotechnika_START:= TRUE;
	ELSIF CasVypnutiaVzduchotechniky.Q THEN
		Linka.OUT.Vzduchotechnika_START:= FALSE;
	END_IF

	CasVypnutiaVzduchotechniky.IN:= Linka.OUT.Vzduchotechnika_START AND NOT Linka.OUT.IonJednotka_START;
	CasVypnutiaVzduchotechniky.PT:= T#30M;
	CasVypnutiaVzduchotechniky();

	//Volanie podprogramov//
	OvlSafety;
	KOM_VentilovyTerminal;
	ZmenaModelu;
	OvlRucnejCitackyQR;

	//****************************************Príznak hardware pracoviska OK***********************************//

	IF StavHardware.KartaAB2_ProfinetMaster_OK AND
		StavHardware.KartaAB3_SafetyMaster_OK AND
		StavHardware.KartaAB4_SafetyDI_OK AND
		StavHardware.KartaAB5_16DI_OK AND
		StavHardware.KartaAB6_16DI_OK AND
		StavHardware.KartaAB7_16DI_OK AND
		StavHardware.KartaAB8_16DO_OK AND
		StavHardware.KartaAB9_16DO_OK AND
		StavHardware.KartaAB10_X2X_OK AND
		StavHardware.ModulDI1_16DI_OK AND
		StavHardware.ModulDI2_16DI_OK AND
		StavHardware.ModulDI3_8DI_OK AND
		StavHardware.ModulSI1_4SI_OK AND
		StavHardware.ModulSI2_4SI_OK AND
		StavHardware.Komunikacia_RFIDModul_OK AND
		StavHardware.Komunikacia_Kamera_OK AND
		StavHardware.Komunikacia_MeniceFM_OK AND
		StavHardware.Komunikacia_Robot_OK AND
		StavHardware.Komunikacia_Panasonic_OK AND
		NOT StavHardware.Komunikacia_VentTerminal_OK THEN
		Linka.STAV.Hardware_OK:= TRUE;
	ELSE
		Linka.STAV.Hardware_OK:= FALSE;
	END_IF

	//***************************************Ovládanie majáka**************************************************//
	//Zelene svetlo//
	IF Linka.STAV.Automat THEN
		Linka.OUT.Majak_ZeleneSvetlo:= TRUE;
	ELSIF Linka.STAV.Manual THEN
		Linka.OUT.Majak_ZeleneSvetlo:= Blikac500ms;
	ELSE
		Linka.OUT.Majak_ZeleneSvetlo:= FALSE;
	END_IF

	//Žlté svetlo//
	IF Linka.STAV.Automat AND NOT Linka.STAV.PoINIT THEN
		Linka.OUT.Majak_ZlteSvetlo:= Blikac500ms;
	ELSIF StoperEtiketovania.STAV.Warning THEN
		Linka.OUT.Majak_ZlteSvetlo:= Blikac500ms;
	ELSE
		Linka.OUT.Majak_ZlteSvetlo:= FALSE;
	END_IF

	//Červené svetlo//
	IF NastalaPorucha THEN
		Linka.OUT.Majak_CerveneSvetlo:= TRUE;
	ELSIF NOT Safety.STAV.ZonaCS_AKTIVNA THEN
		Linka.OUT.Majak_CerveneSvetlo:= TRUE;
	ELSE
		Linka.OUT.Majak_CerveneSvetlo:= FALSE;
	END_IF

	//Húkačka//
	IF EDGEPOS(NastalaPorucha) THEN
		IF CasAktivacieHukacky.Q THEN
			Linka.Majak_HukackaON:= TRUE;
		END_IF
	END_IF

	IF Linka.Majak_HukackaON THEN
		Linka.OUT.Majak_Hukacka:= Blikac500ms;
	ELSE
		Linka.OUT.Majak_Hukacka:= FALSE;
	END_IF

	CasAktivacieHukacky.IN:= NOT Linka.Majak_HukackaON;
	CasAktivacieHukacky.PT:= T#500ms;
	CasAktivacieHukacky();

	//**************************************Ukončenie pracovného cyklu na pracovisku**********************************************//
	//Normálne//
	IF Linka.KoniecCyklu THEN
		VstupVytah.KoniecCyklu:= TRUE;
		StoperPredCistenim.KoniecCyklu:= TRUE;
		StoperPoCisteni.KoniecCyklu:= TRUE;
		DopravCistenia.KoniecCyklu:= TRUE;
		StoperEtiketovania.KoniecCyklu:= TRUE;
		Robot.KoniecCyklu:= TRUE;
		StoperDopravNG.KoniecCyklu:= TRUE;
		DopravBunky.KoniecCyklu:= TRUE;
		StoperVystupDopravnika.KoniecCyklu:= TRUE;
		VystupnyDopravnik.KoniecCyklu:= TRUE;
		VystupVytah.KoniecCyklu:= TRUE;
		StoperVratDopravnika.KoniecCyklu:= TRUE;
		VratnyDopravnik.KoniecCyklu:= TRUE;
		Linka.KoniecCyklu:= FALSE;
	END_IF

	//Pri poruche//
	IF EDGEPOS(PoruchaVstupnehoVytahu) THEN
		VstupVytah.KoniecCyklu:= TRUE;
	END_IF

	IF EDGEPOS(PoruchaCistenia) THEN
		StoperPredCistenim.KoniecCyklu:= TRUE;
		StoperPoCisteni.KoniecCyklu:= TRUE;
		DopravCistenia.KoniecCyklu:= TRUE;
	END_IF

	IF EDGEPOS(PoruchaBunky) THEN
		StoperEtiketovania.KoniecCyklu:= TRUE;
		Robot.KoniecCyklu:= TRUE;
		StoperDopravNG.KoniecCyklu:= TRUE;
		DopravBunky.KoniecCyklu:= TRUE;
	END_IF

	IF EDGEPOS(PoruchaVystupnehoVytahu) THEN
		VystupVytah.KoniecCyklu:= TRUE;
	END_IF

	IF EDGEPOS(PoruchaLinky) THEN
		Linka.KoniecCyklu:= TRUE;
	END_IF

	//Keď dôjde páska v tlačiarni//
	IF Robot.Automat AND StoperEtiketovania.IN.Tlaciaren_KoniecEtikiet THEN
		Vizu.ZobrazHlasenie_DochadzaPaska:= 0;
		Vizu.IndexStavuPasky:= 0;
		StoperEtiketovania.KoniecCyklu:= TRUE;
		Robot.KoniecCyklu:= TRUE;
		StoperDopravNG.KoniecCyklu:= TRUE;
		DopravBunky.KoniecCyklu:= TRUE;
	ELSIF Robot.Automat AND StoperEtiketovania.IN.Tlaciaren_KoniecPasky THEN
		Vizu.ZobrazHlasenie_DochadzaPaska:= 0;
		Vizu.IndexStavuPasky:= 1;
		StoperEtiketovania.KoniecCyklu:= TRUE;
		Robot.KoniecCyklu:= TRUE;
		StoperDopravNG.KoniecCyklu:= TRUE;
		DopravBunky.KoniecCyklu:= TRUE;
	END_IF

	//Status prebieha ukončenie cyklu//
	IF VstupVytah.KoniecCyklu OR
		StoperPredCistenim.KoniecCyklu OR
		StoperPoCisteni.KoniecCyklu OR
		DopravCistenia.KoniecCyklu OR
		StoperEtiketovania.KoniecCyklu OR
		Robot.KoniecCyklu OR
		StoperDopravNG.KoniecCyklu OR
		DopravBunky.KoniecCyklu OR
		StoperVystupDopravnika.KoniecCyklu OR
		VystupnyDopravnik.KoniecCyklu OR
		VystupVytah.KoniecCyklu OR
		StoperVratDopravnika.KoniecCyklu OR
		VratnyDopravnik.KoniecCyklu THEN
		Linka.STAV.UkoncenieCyklu_BUSY:= TRUE;
	ELSE
		Linka.STAV.UkoncenieCyklu_BUSY:= FALSE;
	END_IF

	//****************************************Resetovanie linky****************************************************************//
	//Normálne//
	IF Linka.Reset THEN
		VstupVytah.Reset:= TRUE;
		StoperPredCistenim.Reset:= TRUE;
		StoperPoCisteni.Reset:= TRUE;
		DopravCistenia.Reset:= TRUE;
		StoperEtiketovania.Reset:= TRUE;
		Robot.Reset:= TRUE;
		StoperDopravNG.Reset:= TRUE;
		DopravBunky.Reset:= TRUE;
		StoperVystupDopravnika.Reset:= TRUE;
		VystupnyDopravnik.Reset:= TRUE;
		VystupVytah.Reset:= TRUE;
		StoperVratDopravnika.Reset:= TRUE;
		VratnyDopravnik.Reset:= TRUE;
		Linka.Reset:= FALSE;
	END_IF

	//Pri stlačení tlačítka Automat//
	IF Vizu.TL_RezimAutomat THEN
		IF Linka.STAV.Manual THEN
			Linka.Reset:= TRUE;
		END_IF
		Vizu.TL_RezimAutomat:= FALSE;
	END_IF

	//**************************************Manuálny režim linky*************************************************************//
	IF Linka.Manual THEN
		VstupVytah.Manual:= TRUE;
		StoperPredCistenim.Manual:= TRUE;
		StoperPoCisteni.Manual:= TRUE;
		DopravCistenia.Manual:= TRUE;
		StoperEtiketovania.Manual:= TRUE;
		Robot.Manual:= TRUE;
		StoperDopravNG.Manual:= TRUE;
		DopravBunky.Manual:= TRUE;
		StoperVystupDopravnika.Manual:= TRUE;
		VystupnyDopravnik.Manual:= TRUE;
		VystupVytah.Manual:= TRUE;
		StoperVratDopravnika.Manual:= TRUE;
		VratnyDopravnik.Manual:= TRUE;
		Linka.Manual:= FALSE;
	END_IF

	//Príznak je zvolený režim Manuál//
	IF VstupVytah.Manual OR
		StoperPredCistenim.Manual OR
		StoperPoCisteni.Manual OR
		DopravCistenia.Manual OR
		StoperEtiketovania.Manual OR
		Robot.Manual OR
		StoperDopravNG.Manual OR
		DopravBunky.Manual OR
		StoperVystupDopravnika.Manual OR
		VystupnyDopravnik.Manual OR
		VystupVytah.Manual OR
		StoperVratDopravnika.Manual OR
		VratnyDopravnik.Manual THEN
		Linka.STAV.Manual:= TRUE;
	ELSE
		Linka.STAV.Manual:= FALSE;
	END_IF

	//***************************************Automatický režim pracoviska**********************************************************//
	IF Linka.Automat THEN
		VstupVytah.Automat:= TRUE;
		StoperPredCistenim.Automat:= TRUE;
		StoperPoCisteni.Automat:= TRUE;
		DopravCistenia.Automat:= TRUE;
		StoperEtiketovania.Automat:= TRUE;
		Robot.Automat:= TRUE;
		StoperDopravNG.Automat:= TRUE;
		DopravBunky.Automat:= TRUE;
		StoperVystupDopravnika.Automat:= TRUE;
		VystupnyDopravnik.Automat:= TRUE;
		VystupVytah.Automat:= TRUE;
		StoperVratDopravnika.Automat:= TRUE;
		VratnyDopravnik.Automat:= TRUE;
		Linka.Automat:= FALSE;
	END_IF

	//Príznak je zvolený režim Automat//
	IF VstupVytah.Automat OR
		StoperPredCistenim.Automat OR
		StoperPoCisteni.Automat OR
		DopravCistenia.Automat OR
		StoperEtiketovania.Automat OR
		Robot.Automat OR
		StoperDopravNG.Automat OR
		DopravBunky.Automat OR
		StoperVystupDopravnika.Automat OR
		VystupnyDopravnik.Automat OR
		VystupVytah.Automat OR
		StoperVratDopravnika.Automat OR
		VratnyDopravnik.Automat THEN
		Linka.STAV.Automat:= TRUE;
	ELSE
		Linka.STAV.Automat:= FALSE;
	END_IF

	//Príznak Zariadenie je po inicializácii//
	IF VstupVytah.STAV.PoINIT AND
		StoperPredCistenim.STAV.PoINIT AND
		StoperPoCisteni.STAV.PoINIT AND
		DopravCistenia.STAV.PoINIT AND
		StoperEtiketovania.STAV.PoINIT AND
		Robot.STAV.PoINIT AND
		StoperDopravNG.STAV.PoINIT AND
		DopravBunky.STAV.PoINIT AND
		StoperVystupDopravnika.STAV.PoINIT AND
		VystupnyDopravnik.STAV.PoINIT AND
		VystupVytah.STAV.PoINIT AND
		StoperVratDopravnika.STAV.PoINIT AND
		VratnyDopravnik.STAV.PoINIT THEN
		Linka.STAV.PoINIT:= TRUE;
	ELSE
		Linka.STAV.PoINIT:= FALSE;
	END_IF

	//****************************************Príznak Zariadenie pripravené na spustenie********************************************//
	IF SC_VstupVytah.Step = 1 AND
		SC_StoperPredCistenim.Step = 1 AND
		SC_StoperPoCisteni.Step = 1 AND
		SC_DopravCistenia.Step = 1 AND
		SC_StoperEtiketovania.Step = 1 AND
		SC_Robot.Step = 1 AND
		SC_StoperDopravNG.Step = 1 AND
		SC_DopravBunky.Step = 1 AND
		SC_StoperVystupDopravnika.Step = 1 AND
		SC_VystupnyDopravnik.Step = 1 AND
		SC_VystupVytah.Step = 1 AND
		SC_StoperVratDopravnika.Step = 1 AND
		SC_VratnyDopravnik.Step = 1 THEN
		Linka.STAV.READY_TO_START:= TRUE;
	ELSE
		Linka.STAV.READY_TO_START:= FALSE;
	END_IF

	//******************************************Pauza dopravníkov linky**************************************************************//

	IF Linka.STAV.Automat AND
		NOT VstupVytah.OUT.Dopravnik_ChodVPRED_ELR1 AND
		NOT VstupVytah.OUT.Dopravnik_ChodVZAD_ELR1 AND
		NOT StoperPredCistenim.OUT.StoperZASUN_YV005 AND
		NOT StoperPoCisteni.OUT.StoperZASUN_YV006 AND
		NOT StoperEtiketovania.OUT.StoperZASUN_YV007 AND
		NOT StoperDopravNG.OUT.Dopravnik_ChodVZAD_ELR3 AND
		NOT StoperVystupDopravnika.OUT.StoperZASUN_YV011 AND
		NOT VystupVytah.OUT.Dopravnik_ChodVPRED_ELR6 AND
		NOT VystupVytah.OUT.Dopravnik_ChodVZAD_ELR6 AND
		NOT StoperVratDopravnika.OUT.StoperZASUN_YV012 THEN
		CasDoPauzyDopravnikov.IN:= TRUE;
	ELSE
		CasDoPauzyDopravnikov.IN:= FALSE;
	END_IF

	Linka.STAV.Dopravniky_PAUZA:= CasDoPauzyDopravnikov.Q;

	CasDoPauzyDopravnikov.PT:= T#3M;
	CasDoPauzyDopravnikov();

END_PROGRAM

PROGRAM _EXIT
	(* Insert code here *)

END_PROGRAM
```

#### Variables.var - Local variables
```iecst
VAR
	CasResetZonyVstupVytahu : TON;
	CasResetZonyBunky : TON;
	CasResetZonyVystupVytahu : TON;
	SC_ZmenaModelu : SequenceControlTyp := (0);
	i : USINT := 0;
	ModelNajdeny : BOOL := FALSE;
	Nacitany_LOT_POLE : ARRAY[0..10] OF USINT := [11(0)];
	PocetNacitanychZnakov : UDINT := 0;
	NacitaneZnaky_POLE : ARRAY[0..100] OF USINT := [101(0)];
	a : UINT := 0;
	CasAktivacieHukacky : TON := (0);
	CasVypnutiaVzduchotechniky : TON := (0);
	CasDoPauzyDopravnikov : TON := (0);
END_VAR
```

#### OvlSafety.st
```iecst
ACTION OvlSafety:

	//Podsvietenie tlačítka Reset CS//
	IF Safety.STAV.CS_OvlPanel_Odblokovany AND Safety.STAV.CS_Robot_Odblokovany AND Safety.STAV.CS_VstupnyVytah_Odblokovany AND Safety.STAV.CS_VystupnyVytah_Odblokovany AND NOT Safety.STAV.ZonaCS_AKTIVNA THEN
		Vizu.PodsvietenieTlacitka_ResetCS:= Blikac500ms;
	ELSIF Safety.STAV.ZonaCS_AKTIVNA THEN
		Vizu.PodsvietenieTlacitka_ResetCS:= 2;
	ELSE
		Vizu.PodsvietenieTlacitka_ResetCS:= 3;
	END_IF

	//Podsvietenie tlačítok zámkov dverí//
	//Predné dvere//
	IF Linka.IN.PredneDvereZavrete_EZ1 AND NOT Linka.OUT.PredneDvere_Zamkni_EZ1 THEN
		Vizu.FarbaTlacitka_ZamokPredneDvere:= Blikac500ms;
	ELSIF Linka.IN.PredneDvereZavrete_EZ1 AND Linka.OUT.PredneDvere_Zamkni_EZ1 THEN
		Vizu.FarbaTlacitka_ZamokPredneDvere:= 2;
	ELSE
		Vizu.FarbaTlacitka_ZamokPredneDvere:= 3;
	END_IF

	//Zadné dvere//
	IF Linka.IN.ZadneDvereZavrete_EZ2 AND NOT Linka.OUT.ZadneDvere_Zamkni_EZ2 THEN
		Vizu.FarbaTlacitka_ZamokZadneDvere:= Blikac500ms;
	ELSIF Linka.IN.ZadneDvereZavrete_EZ2 AND Linka.OUT.ZadneDvere_Zamkni_EZ2 THEN
		Vizu.FarbaTlacitka_ZamokZadneDvere:= 2;
	ELSE
		Vizu.FarbaTlacitka_ZamokZadneDvere:= 3;
	END_IF

	//******************************************Ovládanie zámkov dverí bunky****************************************//
	//Predné dvere //
	IF Vizu.TL_ZamkniPredneDvere THEN
		IF Linka.IN.PredneDvereZavrete_EZ1 THEN
			IF Linka.OUT.PredneDvere_Zamkni_EZ1 THEN
				Linka.OUT.PredneDvere_Zamkni_EZ1:= FALSE;
			ELSE
				Linka.OUT.PredneDvere_Zamkni_EZ1:= TRUE;
			END_IF
		END_IF
		Vizu.TL_ZamkniPredneDvere:= FALSE;
	END_IF

	//Zadné dvere //
	IF Vizu.TL_ZamkniZadneDvere THEN
		IF Linka.IN.ZadneDvereZavrete_EZ2 THEN
			IF Linka.OUT.ZadneDvere_Zamkni_EZ2 THEN
				Linka.OUT.ZadneDvere_Zamkni_EZ2:= FALSE;
			ELSE
				Linka.OUT.ZadneDvere_Zamkni_EZ2:= TRUE;
			END_IF
		END_IF
		Vizu.TL_ZamkniZadneDvere:= FALSE;
	END_IF

	//************************************************Resetovanie zón****************************************************//
	//Reset zóny vstupného výťahu//
	CasResetZonyVstupVytahu.IN:= NOT Safety.STAV.ZonaVstupnyVytah_AKTIVNA AND Safety.STAV.ZonaVstupnyVytah_Odblokovana;

	IF CasResetZonyVstupVytahu.Q THEN
		Safety.RESET_ZonyVstupnehoVytahu:= TRUE;
	ELSE
		Safety.RESET_ZonyVstupnehoVytahu:= FALSE;
	END_IF

	CasResetZonyVstupVytahu.PT:= T#1s;
	CasResetZonyVstupVytahu();

	//Reset zóny bunky//
	CasResetZonyBunky.IN:= NOT Safety.STAV.ZonaBunky_AKTIVNA AND Safety.STAV.ZonaBunky_Odblokovana;

	IF CasResetZonyBunky.Q THEN
		Safety.RESET_ZonyBunky:= TRUE;
	ELSE
		Safety.RESET_ZonyBunky:= FALSE;
	END_IF

	CasResetZonyBunky.PT:= T#1s;
	CasResetZonyBunky();

	//Reset zóny výstupného výťahu//
	CasResetZonyVystupVytahu.IN:= NOT Safety.STAV.ZonaVystupnyVytah_AKTIVNA AND Safety.STAV.ZonaVystupnyVytah_Odblokovana;

	IF CasResetZonyVystupVytahu.Q THEN
		Safety.RESET_ZonyVystupnehoVytahu:= TRUE;
	ELSE
		Safety.RESET_ZonyVystupnehoVytahu:= FALSE;
	END_IF

	CasResetZonyVystupVytahu.PT:= T#1s;
	CasResetZonyVystupVytahu();

	//Reset dedman//
	IF NOT Linka.STAV.Automat AND ZvolenaUroven > 30 AND Safety.STAV.DeadMan_Odblokovany AND NOT Safety.STAV.DeadMan_AKTIVNY THEN
		Safety.RESET_DeadMan:= TRUE;
	ELSE
		Safety.RESET_DeadMan:= FALSE;
	END_IF

END_ACTION
```

#### KOM_VentilTerminal.st
```iecst
ACTION KOM_VentilovyTerminal:

	//Mapovanie ventilového terminálu VT1//

//	Linka.OUT.VT1_PowerlinkOUTPUTS[0].0;
//	Linka.OUT.VT1_PowerlinkOUTPUTS[0].1;
//	Linka.OUT.VT1_PowerlinkOUTPUTS[0].2:= VstupVytah.OUT.DvereVytahu_ZATVOR_YV001;
//	Linka.OUT.VT1_PowerlinkOUTPUTS[0].3:= VstupVytah.OUT.DvereVytahu_OTVOR_YV002;
//	Linka.OUT.VT1_PowerlinkOUTPUTS[0].4;
//	Linka.OUT.VT1_PowerlinkOUTPUTS[0].5;
//	Linka.OUT.VT1_PowerlinkOUTPUTS[0].6:= StoperEtiketovania.OUT.Centrovanie_VYSUN_YV003;
//	Linka.OUT.VT1_PowerlinkOUTPUTS[0].7:= StoperEtiketovania.OUT.Centrovanie_ZASUN_YV004;
//
//
//	Linka.OUT.VT1_PowerlinkOUTPUTS[1].0:= StoperPredCistenim.OUT.StoperZASUN_YV005;
//	Linka.OUT.VT1_PowerlinkOUTPUTS[1].1:= StoperPoCisteni.OUT.StoperZASUN_YV006;
//	Linka.OUT.VT1_PowerlinkOUTPUTS[1].2:= StoperEtiketovania.OUT.StoperZASUN_YV007;
//	Linka.OUT.VT1_PowerlinkOUTPUTS[1].3:= StoperDopravNG.OUT.NatlakujTlmicPaletky_YV008;
//	Linka.OUT.VT1_PowerlinkOUTPUTS[1].4:= StoperDopravNG.OUT.Centrovanie_VYSUN_YV009;
//	Linka.OUT.VT1_PowerlinkOUTPUTS[1].5:= StoperDopravNG.OUT.Centrovanie_ZASUN_YV010;
//	Linka.OUT.VT1_PowerlinkOUTPUTS[1].6:= StoperVystupDopravnika.OUT.StoperZASUN_YV011;
//	Linka.OUT.VT1_PowerlinkOUTPUTS[1].7:= StoperVratDopravnika.OUT.StoperZASUN_YV012;
//
//
//	Linka.OUT.VT1_PowerlinkOUTPUTS[2].0;
//	Linka.OUT.VT1_PowerlinkOUTPUTS[2].1;
//	Linka.OUT.VT1_PowerlinkOUTPUTS[2].2:= Robot.OUT.PrisavanieEtikety_ZAPNI_YV013;
//	Linka.OUT.VT1_PowerlinkOUTPUTS[2].3:= Robot.OUT.PrisavanieEtikety_VYPNI_YV014;
//	Linka.OUT.VT1_PowerlinkOUTPUTS[2].4;
//	Linka.OUT.VT1_PowerlinkOUTPUTS[2].5;
//	Linka.OUT.VT1_PowerlinkOUTPUTS[2].6;
//	Linka.OUT.VT1_PowerlinkOUTPUTS[2].7;

END_ACTION
```
